KUKA KRL program: CIRCULO10X10_00.src

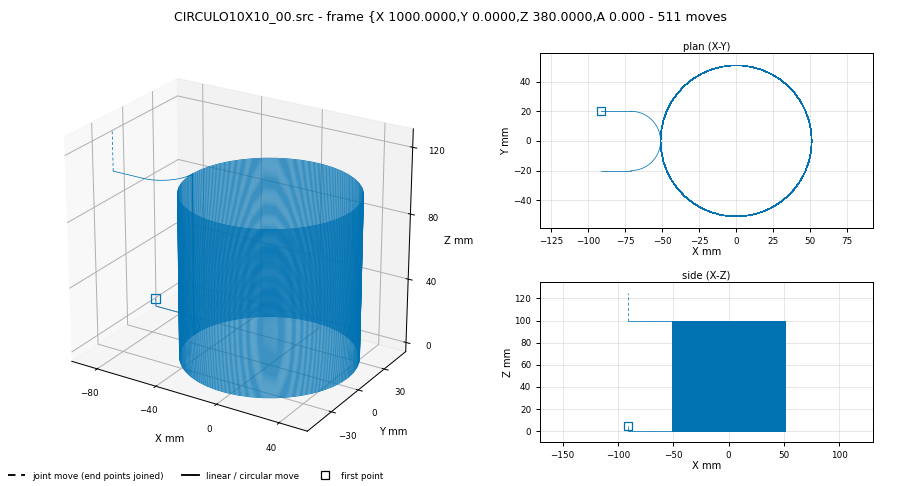
[picture p0: tool path of CIRCULO10X10_00.src in frame {X 1000.0000,Y 0.0000,Z 380.0000,A 0.000, 511 of 513 moves have a stored position in this frame; points joined in program order, loops and branches not executed]
&ACCESS RVP
&REL 1
&COMMENT GENERATED BY ROBOTMASTER
&PARAM TEMPLATE = C:\KRC\Roboter\Template\vorgabe
&PARAM EDITMASK = *
DEF CIRCULO10X2_00()

EXT BAS (BAS_COMMAND :IN,REAL :IN )

INT I

BAS (#INITMOV,0 )

;******SETTINGS FOR PTP MOTION***********************
;FOLD
;SET PTP $VEL_AXIS AND $ACC_AXIS
FOR I=1 TO 6
   $VEL_AXIS[I]=50
   $ACC_AXIS[I]=100
ENDFOR
;ENDFOLD (SET PTP $VEL_AXIS AND $ACC_AXIS)

;******SETTINGS FOR LIN AND ARC MOTION***************
;FOLD
;SET LIN AND ARC MOTION VARIABLES
$VEL.CP=0.262059
$VEL.ORI1=200
$VEL.ORI2=200
$ACC.ORI1=100
$ACC.ORI2=100
;ENDFOLD (SET LIN AND ARC MOTION VARIABLES)

;******SETTINGS FOR POSITIONING CRITERIA*************
;FOLD
;SET POSITIONING CRITERIA
  $APO.CDIS = 0.5000
  $ORI_TYPE = #VAR
;ENDFOLD (SET POSITIONING CRITERIA)

$BASE={X 1000.0000,Y 0.0000,Z 380.0000,A 0.0000,B 0.0000,C 0.0000}
$TOOL={X 63.3526,Y -0.0008,Z 236.7470,A 0.0000,B 30.5004,C 0.0000}

$ADVANCE = 5
PTP  {A1 20.0000,A2 -90.0000,A3 90.0000,A4 0.0000,A5 45.0000,A6 0.0000}
PTP  {X -91.0000,Y 20.0000,Z 5.0000,A 180.0000,B 0.0000,C 180.0000,S 2,T 35}
PTP  {X -91.0000,Y 20.0000,Z 2.0000,A 180.0000,B 0.0000,C 180.0000,S 2,T 35}
$VEL.CP=0.1  ;100mm/s
LIN  {X -91.0000,Y 20.0000,Z 0.0000,A 180.0000,B 0.0000,C 180.0000} C_DIS
LIN  {X -71.0000,Y 20.0000,Z 0.0000,A 180.0000,B 0.0000,C 180.0000} C_DIS
CIRC {X -56.8579,Y 14.1421,Z 0.0000,A 180.0000,B 0.0000,C 180.0000},{X -51.0000,Y 0.0000,Z 0.0000,A 180.0000,B 0.0000,C 180.0000} C_DIS
CIRC {X 0.0000,Y -51.0000,Z 0.0000,A 180.0000,B 0.0000,C 180.0000},{X 51.0000,Y 0.0000,Z 0.0000,A 180.0000,B 0.0000,C 180.0000} C_DIS
CIRC {X 0.0000,Y 51.0000,Z 0.0000,A 180.0000,B 0.0000,C 180.0000},{X -51.0000,Y 0.0000,Z 0.0000,A 180.0000,B 0.0000,C 180.0000} C_DIS
LIN  {X -51.0000,Y 0.0000,Z 0.5970,A 180.0000,B 0.0000,C 180.0000} C_DIS
CIRC {X 0.0000,Y -51.0000,Z 0.5970,A 180.0000,B 0.0000,C 180.0000},{X 51.0000,Y 0.0000,Z 0.5970,A 180.0000,B 0.0000,C 180.0000} C_DIS
CIRC {X 0.0000,Y 51.0000,Z 0.5970,A 180.0000,B 0.0000,C 180.0000},{X -51.0000,Y 0.0000,Z 0.5970,A 180.0000,B 0.0000,C 180.0000} C_DIS
LIN  {X -51.0000,Y 0.0000,Z 1.1976,A 180.0000,B 0.0000,C 180.0000} C_DIS
CIRC {X 0.0000,Y -51.0000,Z 1.1976,A 180.0000,B 0.0000,C 180.0000},{X 51.0000,Y 0.0000,Z 1.1976,A 180.0000,B 0.0000,C 180.0000} C_DIS
CIRC {X 0.0000,Y 51.0000,Z 1.1976,A 180.0000,B 0.0000,C 180.0000},{X -51.0000,Y 0.0000,Z 1.1976,A 180.0000,B 0.0000,C 180.0000} C_DIS
LIN  {X -51.0000,Y 0.0000,Z 1.7964,A 180.0000,B 0.0000,C 180.0000} C_DIS
CIRC {X 0.0000,Y -51.0000,Z 1.7964,A 180.0000,B 0.0000,C 180.0000},{X 51.0000,Y 0.0000,Z 1.7964,A 180.0000,B 0.0000,C 180.0000} C_DIS
CIRC {X 0.0000,Y 51.0000,Z 1.7964,A 180.0000,B 0.0000,C 180.0000},{X -51.0000,Y 0.0000,Z 1.7964,A 180.0000,B 0.0000,C 180.0000} C_DIS
LIN  {X -51.0000,Y 0.0000,Z 2.3952,A 180.0000,B 0.0000,C 180.0000} C_DIS
CIRC {X 0.0000,Y -51.0000,Z 2.3952,A 180.0000,B 0.0000,C 180.0000},{X 51.0000,Y 0.0000,Z 2.3952,A 180.0000,B 0.0000,C 180.0000} C_DIS
CIRC {X 0.0000,Y 51.0000,Z 2.3952,A 180.0000,B 0.0000,C 180.0000},{X -51.0000,Y 0.0000,Z 2.3952,A 180.0000,B 0.0000,C 180.0000} C_DIS
LIN  {X -51.0000,Y 0.0000,Z 2.9940,A 180.0000,B 0.0000,C 180.0000} C_DIS
CIRC {X 0.0000,Y -51.0000,Z 2.9940,A 180.0000,B 0.0000,C 180.0000},{X 51.0000,Y 0.0000,Z 2.9940,A 180.0000,B 0.0000,C 180.0000} C_DIS
CIRC {X 0.0000,Y 51.0000,Z 2.9940,A 180.0000,B 0.0000,C 180.0000},{X -51.0000,Y 0.0000,Z 2.9940,A 180.0000,B 0.0000,C 180.0000} C_DIS
LIN  {X -51.0000,Y 0.0000,Z 3.5928,A 180.0000,B 0.0000,C 180.0000} C_DIS
CIRC {X 0.0000,Y -51.0000,Z 3.5928,A 180.0000,B 0.0000,C 180.0000},{X 51.0000,Y 0.0000,Z 3.5928,A 180.0000,B 0.0000,C 180.0000} C_DIS
CIRC {X 0.0000,Y 51.0000,Z 3.5928,A 180.0000,B 0.0000,C 180.0000},{X -51.0000,Y 0.0000,Z 3.5928,A 180.0000,B 0.0000,C 180.0000} C_DIS
LIN  {X -51.0000,Y 0.0000,Z 4.1916,A 180.0000,B 0.0000,C 180.0000} C_DIS
CIRC {X 0.0000,Y -51.0000,Z 4.1916,A 180.0000,B 0.0000,C 180.0000},{X 51.0000,Y 0.0000,Z 4.1916,A 180.0000,B 0.0000,C 180.0000} C_DIS
CIRC {X 0.0000,Y 51.0000,Z 4.1916,A 180.0000,B 0.0000,C 180.0000},{X -51.0000,Y 0.0000,Z 4.1916,A 180.0000,B 0.0000,C 180.0000} C_DIS
LIN  {X -51.0000,Y 0.0000,Z 4.7904,A 180.0000,B 0.0000,C 180.0000} C_DIS
CIRC {X 0.0000,Y -51.0000,Z 4.7904,A 180.0000,B 0.0000,C 180.0000},{X 51.0000,Y 0.0000,Z 4.7904,A 180.0000,B 0.0000,C 180.0000} C_DIS
CIRC {X 0.0000,Y 51.0000,Z 4.7904,A 180.0000,B 0.0000,C 180.0000},{X -51.0000,Y 0.0000,Z 4.7904,A 180.0000,B 0.0000,C 180.0000} C_DIS
LIN  {X -51.0000,Y 0.0000,Z 5.3892,A 180.0000,B 0.0000,C 180.0000} C_DIS
CIRC {X 0.0000,Y -51.0000,Z 5.3892,A 180.0000,B 0.0000,C 180.0000},{X 51.0000,Y 0.0000,Z 5.3892,A 180.0000,B 0.0000,C 180.0000} C_DIS
CIRC {X 0.0000,Y 51.0000,Z 5.3892,A 180.0000,B 0.0000,C 180.0000},{X -51.0000,Y 0.0000,Z 5.3892,A 180.0000,B 0.0000,C 180.0000} C_DIS
LIN  {X -51.0000,Y 0.0000,Z 5.9880,A 180.0000,B 0.0000,C 180.0000} C_DIS
CIRC {X 0.0000,Y -51.0000,Z 5.9880,A 180.0000,B 0.0000,C 180.0000},{X 51.0000,Y 0.0000,Z 5.9880,A 180.0000,B 0.0000,C 180.0000} C_DIS
CIRC {X 0.0000,Y 51.0000,Z 5.9880,A 180.0000,B 0.0000,C 180.0000},{X -51.0000,Y 0.0000,Z 5.9880,A 180.0000,B 0.0000,C 180.0000} C_DIS
LIN  {X -51.0000,Y 0.0000,Z 6.5868,A 180.0000,B 0.0000,C 180.0000} C_DIS
CIRC {X 0.0000,Y -51.0000,Z 6.5868,A 180.0000,B 0.0000,C 180.0000},{X 51.0000,Y 0.0000,Z 6.5868,A 180.0000,B 0.0000,C 180.0000} C_DIS
CIRC {X 0.0000,Y 51.0000,Z 6.5868,A 180.0000,B 0.0000,C 180.0000},{X -51.0000,Y 0.0000,Z 6.5868,A 180.0000,B 0.0000,C 180.0000} C_DIS
LIN  {X -51.0000,Y 0.0000,Z 7.1856,A 180.0000,B 0.0000,C 180.0000} C_DIS
CIRC {X 0.0000,Y -51.0000,Z 7.1856,A 180.0000,B 0.0000,C 180.0000},{X 51.0000,Y 0.0000,Z 7.1856,A 180.0000,B 0.0000,C 180.0000} C_DIS
CIRC {X 0.0000,Y 51.0000,Z 7.1856,A 180.0000,B 0.0000,C 180.0000},{X -51.0000,Y 0.0000,Z 7.1856,A 180.0000,B 0.0000,C 180.0000} C_DIS
LIN  {X -51.0000,Y 0.0000,Z 7.7844,A 180.0000,B 0.0000,C 180.0000} C_DIS
CIRC {X 0.0000,Y -51.0000,Z 7.7844,A 180.0000,B 0.0000,C 180.0000},{X 51.0000,Y 0.0000,Z 7.7844,A 180.0000,B 0.0000,C 180.0000} C_DIS
CIRC {X 0.0000,Y 51.0000,Z 7.7844,A 180.0000,B 0.0000,C 180.0000},{X -51.0000,Y 0.0000,Z 7.7844,A 180.0000,B 0.0000,C 180.0000} C_DIS
LIN  {X -51.0000,Y 0.0000,Z 8.3832,A 180.0000,B 0.0000,C 180.0000} C_DIS
CIRC {X 0.0000,Y -51.0000,Z 8.3832,A 180.0000,B 0.0000,C 180.0000},{X 51.0000,Y 0.0000,Z 8.3832,A 180.0000,B 0.0000,C 180.0000} C_DIS
CIRC {X 0.0000,Y 51.0000,Z 8.3832,A 180.0000,B 0.0000,C 180.0000},{X -51.0000,Y 0.0000,Z 8.3832,A 180.0000,B 0.0000,C 180.0000} C_DIS
LIN  {X -51.0000,Y 0.0000,Z 8.9820,A 180.0000,B 0.0000,C 180.0000} C_DIS
CIRC {X 0.0000,Y -51.0000,Z 8.9820,A 180.0000,B 0.0000,C 180.0000},{X 51.0000,Y 0.0000,Z 8.9820,A 180.0000,B 0.0000,C 180.0000} C_DIS
CIRC {X 0.0000,Y 51.0000,Z 8.9820,A 180.0000,B 0.0000,C 180.0000},{X -51.0000,Y 0.0000,Z 8.9820,A 180.0000,B 0.0000,C 180.0000} C_DIS
LIN  {X -51.0000,Y 0.0000,Z 9.5808,A 180.0000,B 0.0000,C 180.0000} C_DIS
CIRC {X 0.0000,Y -51.0000,Z 9.5808,A 180.0000,B 0.0000,C 180.0000},{X 51.0000,Y 0.0000,Z 9.5808,A 180.0000,B 0.0000,C 180.0000} C_DIS
CIRC {X 0.0000,Y 51.0000,Z 9.5808,A 180.0000,B 0.0000,C 180.0000},{X -51.0000,Y 0.0000,Z 9.5808,A 180.0000,B 0.0000,C 180.0000} C_DIS
LIN  {X -51.0000,Y 0.0000,Z 10.1796,A 180.0000,B 0.0000,C 180.0000} C_DIS
CIRC {X 0.0000,Y -51.0000,Z 10.1796,A 180.0000,B 0.0000,C 180.0000},{X 51.0000,Y 0.0000,Z 10.1796,A 180.0000,B 0.0000,C 180.0000} C_DIS
CIRC {X 0.0000,Y 51.0000,Z 10.1796,A 180.0000,B 0.0000,C 180.0000},{X -51.0000,Y 0.0000,Z 10.1796,A 180.0000,B 0.0000,C 180.0000} C_DIS
LIN  {X -51.0000,Y 0.0000,Z 10.7784,A 180.0000,B 0.0000,C 180.0000} C_DIS
CIRC {X 0.0000,Y -51.0000,Z 10.7784,A 180.0000,B 0.0000,C 180.0000},{X 51.0000,Y 0.0000,Z 10.7784,A 180.0000,B 0.0000,C 180.0000} C_DIS
CIRC {X 0.0000,Y 51.0000,Z 10.7784,A 180.0000,B 0.0000,C 180.0000},{X -51.0000,Y 0.0000,Z 10.7784,A 180.0000,B 0.0000,C 180.0000} C_DIS
LIN  {X -51.0000,Y 0.0000,Z 11.3772,A 180.0000,B 0.0000,C 180.0000} C_DIS
CIRC {X 0.0000,Y -51.0000,Z 11.3772,A 180.0000,B 0.0000,C 180.0000},{X 51.0000,Y 0.0000,Z 11.3772,A 180.0000,B 0.0000,C 180.0000} C_DIS
CIRC {X 0.0000,Y 51.0000,Z 11.3772,A 180.0000,B 0.0000,C 180.0000},{X -51.0000,Y 0.0000,Z 11.3772,A 180.0000,B 0.0000,C 180.0000} C_DIS
LIN  {X -51.0000,Y 0.0000,Z 11.9760,A 180.0000,B 0.0000,C 180.0000} C_DIS
CIRC {X 0.0000,Y -51.0000,Z 11.9760,A 180.0000,B 0.0000,C 180.0000},{X 51.0000,Y 0.0000,Z 11.9760,A 180.0000,B 0.0000,C 180.0000} C_DIS
CIRC {X 0.0000,Y 51.0000,Z 11.9760,A 180.0000,B 0.0000,C 180.0000},{X -51.0000,Y 0.0000,Z 11.9760,A 180.0000,B 0.0000,C 180.0000} C_DIS
LIN  {X -51.0000,Y 0.0000,Z 12.5748,A 180.0000,B 0.0000,C 180.0000} C_DIS
CIRC {X 0.0000,Y -51.0000,Z 12.5748,A 180.0000,B 0.0000,C 180.0000},{X 51.0000,Y 0.0000,Z 12.5748,A 180.0000,B 0.0000,C 180.0000} C_DIS
CIRC {X 0.0000,Y 51.0000,Z 12.5748,A 180.0000,B 0.0000,C 180.0000},{X -51.0000,Y 0.0000,Z 12.5748,A 180.0000,B 0.0000,C 180.0000} C_DIS
LIN  {X -51.0000,Y 0.0000,Z 13.1737,A 180.0000,B 0.0000,C 180.0000} C_DIS
CIRC {X 0.0000,Y -51.0000,Z 13.1737,A 180.0000,B 0.0000,C 180.0000},{X 51.0000,Y 0.0000,Z 13.1737,A 180.0000,B 0.0000,C 180.0000} C_DIS
CIRC {X 0.0000,Y 51.0000,Z 13.1737,A 180.0000,B 0.0000,C 180.0000},{X -51.0000,Y 0.0000,Z 13.1737,A 180.0000,B 0.0000,C 180.0000} C_DIS
LIN  {X -51.0000,Y 0.0000,Z 13.7725,A 180.0000,B 0.0000,C 180.0000} C_DIS
CIRC {X 0.0000,Y -51.0000,Z 13.7725,A 180.0000,B 0.0000,C 180.0000},{X 51.0000,Y 0.0000,Z 13.7725,A 180.0000,B 0.0000,C 180.0000} C_DIS
CIRC {X 0.0000,Y 51.0000,Z 13.7725,A 180.0000,B 0.0000,C 180.0000},{X -51.0000,Y 0.0000,Z 13.7725,A 180.0000,B 0.0000,C 180.0000} C_DIS
LIN  {X -51.0000,Y 0.0000,Z 14.3713,A 180.0000,B 0.0000,C 180.0000} C_DIS
CIRC {X 0.0000,Y -51.0000,Z 14.3713,A 180.0000,B 0.0000,C 180.0000},{X 51.0000,Y 0.0000,Z 14.3713,A 180.0000,B 0.0000,C 180.0000} C_DIS
CIRC {X 0.0000,Y 51.0000,Z 14.3713,A 180.0000,B 0.0000,C 180.0000},{X -51.0000,Y 0.0000,Z 14.3713,A 180.0000,B 0.0000,C 180.0000} C_DIS
LIN  {X -51.0000,Y 0.0000,Z 14.9701,A 180.0000,B 0.0000,C 180.0000} C_DIS
CIRC {X 0.0000,Y -51.0000,Z 14.9701,A 180.0000,B 0.0000,C 180.0000},{X 51.0000,Y 0.0000,Z 14.9701,A 180.0000,B 0.0000,C 180.0000} C_DIS
CIRC {X 0.0000,Y 51.0000,Z 14.9701,A 180.0000,B 0.0000,C 180.0000},{X -51.0000,Y 0.0000,Z 14.9701,A 180.0000,B 0.0000,C 180.0000} C_DIS
LIN  {X -51.0000,Y 0.0000,Z 15.5689,A 180.0000,B 0.0000,C 180.0000} C_DIS
CIRC {X 0.0000,Y -51.0000,Z 15.5689,A 180.0000,B 0.0000,C 180.0000},{X 51.0000,Y 0.0000,Z 15.5689,A 180.0000,B 0.0000,C 180.0000} C_DIS
CIRC {X 0.0000,Y 51.0000,Z 15.5689,A 180.0000,B 0.0000,C 180.0000},{X -51.0000,Y 0.0000,Z 15.5689,A 180.0000,B 0.0000,C 180.0000} C_DIS
LIN  {X -51.0000,Y 0.0000,Z 16.1677,A 180.0000,B 0.0000,C 180.0000} C_DIS
CIRC {X 0.0000,Y -51.0000,Z 16.1677,A 180.0000,B 0.0000,C 180.0000},{X 51.0000,Y 0.0000,Z 16.1677,A 180.0000,B 0.0000,C 180.0000} C_DIS
CIRC {X 0.0000,Y 51.0000,Z 16.1677,A 180.0000,B 0.0000,C 180.0000},{X -51.0000,Y 0.0000,Z 16.1677,A 180.0000,B 0.0000,C 180.0000} C_DIS
LIN  {X -51.0000,Y 0.0000,Z 16.7665,A 180.0000,B 0.0000,C 180.0000} C_DIS
CIRC {X 0.0000,Y -51.0000,Z 16.7665,A 180.0000,B 0.0000,C 180.0000},{X 51.0000,Y 0.0000,Z 16.7665,A 180.0000,B 0.0000,C 180.0000} C_DIS
CIRC {X 0.0000,Y 51.0000,Z 16.7665,A 180.0000,B 0.0000,C 180.0000},{X -51.0000,Y 0.0000,Z 16.7665,A 180.0000,B 0.0000,C 180.0000} C_DIS
LIN  {X -51.0000,Y 0.0000,Z 17.3653,A 180.0000,B 0.0000,C 180.0000} C_DIS
CIRC {X 0.0000,Y -51.0000,Z 17.3653,A 180.0000,B 0.0000,C 180.0000},{X 51.0000,Y 0.0000,Z 17.3653,A 180.0000,B 0.0000,C 180.0000} C_DIS
CIRC {X 0.0000,Y 51.0000,Z 17.3653,A 180.0000,B 0.0000,C 180.0000},{X -51.0000,Y 0.0000,Z 17.3653,A 180.0000,B 0.0000,C 180.0000} C_DIS
LIN  {X -51.0000,Y 0.0000,Z 17.9641,A 180.0000,B 0.0000,C 180.0000} C_DIS
CIRC {X 0.0000,Y -51.0000,Z 17.9641,A 180.0000,B 0.0000,C 180.0000},{X 51.0000,Y 0.0000,Z 17.9641,A 180.0000,B 0.0000,C 180.0000} C_DIS
CIRC {X 0.0000,Y 51.0000,Z 17.9641,A 180.0000,B 0.0000,C 180.0000},{X -51.0000,Y 0.0000,Z 17.9641,A 180.0000,B 0.0000,C 180.0000} C_DIS
LIN  {X -51.0000,Y 0.0000,Z 18.5629,A 180.0000,B 0.0000,C 180.0000} C_DIS
CIRC {X 0.0000,Y -51.0000,Z 18.5629,A 180.0000,B 0.0000,C 180.0000},{X 51.0000,Y 0.0000,Z 18.5629,A 180.0000,B 0.0000,C 180.0000} C_DIS
CIRC {X 0.0000,Y 51.0000,Z 18.5629,A 180.0000,B 0.0000,C 180.0000},{X -51.0000,Y 0.0000,Z 18.5629,A 180.0000,B 0.0000,C 180.0000} C_DIS
LIN  {X -51.0000,Y 0.0000,Z 19.1617,A 180.0000,B 0.0000,C 180.0000} C_DIS
CIRC {X 0.0000,Y -51.0000,Z 19.1617,A 180.0000,B 0.0000,C 180.0000},{X 51.0000,Y 0.0000,Z 19.1617,A 180.0000,B 0.0000,C 180.0000} C_DIS
CIRC {X 0.0000,Y 51.0000,Z 19.1617,A 180.0000,B 0.0000,C 180.0000},{X -51.0000,Y 0.0000,Z 19.1617,A 180.0000,B 0.0000,C 180.0000} C_DIS
LIN  {X -51.0000,Y 0.0000,Z 19.7605,A 180.0000,B 0.0000,C 180.0000} C_DIS
CIRC {X 0.0000,Y -51.0000,Z 19.7605,A 180.0000,B 0.0000,C 180.0000},{X 51.0000,Y 0.0000,Z 19.7605,A 180.0000,B 0.0000,C 180.0000} C_DIS
CIRC {X 0.0000,Y 51.0000,Z 19.7605,A 180.0000,B 0.0000,C 180.0000},{X -51.0000,Y 0.0000,Z 19.7605,A 180.0000,B 0.0000,C 180.0000} C_DIS
LIN  {X -51.0000,Y 0.0000,Z 20.3593,A 180.0000,B 0.0000,C 180.0000} C_DIS
CIRC {X 0.0000,Y -51.0000,Z 20.3593,A 180.0000,B 0.0000,C 180.0000},{X 51.0000,Y 0.0000,Z 20.3593,A 180.0000,B 0.0000,C 180.0000} C_DIS
CIRC {X 0.0000,Y 51.0000,Z 20.3593,A 180.0000,B 0.0000,C 180.0000},{X -51.0000,Y 0.0000,Z 20.3593,A 180.0000,B 0.0000,C 180.0000} C_DIS
LIN  {X -51.0000,Y 0.0000,Z 20.9581,A 180.0000,B 0.0000,C 180.0000} C_DIS
CIRC {X 0.0000,Y -51.0000,Z 20.9581,A 180.0000,B 0.0000,C 180.0000},{X 51.0000,Y 0.0000,Z 20.9581,A 180.0000,B 0.0000,C 180.0000} C_DIS
CIRC {X 0.0000,Y 51.0000,Z 20.9581,A 180.0000,B 0.0000,C 180.0000},{X -51.0000,Y 0.0000,Z 20.9581,A 180.0000,B 0.0000,C 180.0000} C_DIS
LIN  {X -51.0000,Y 0.0000,Z 21.5569,A 180.0000,B 0.0000,C 180.0000} C_DIS
CIRC {X 0.0000,Y -51.0000,Z 21.5569,A 180.0000,B 0.0000,C 180.0000},{X 51.0000,Y 0.0000,Z 21.5569,A 180.0000,B 0.0000,C 180.0000} C_DIS
CIRC {X 0.0000,Y 51.0000,Z 21.5569,A 180.0000,B 0.0000,C 180.0000},{X -51.0000,Y 0.0000,Z 21.5569,A 180.0000,B 0.0000,C 180.0000} C_DIS
LIN  {X -51.0000,Y 0.0000,Z 22.1557,A 180.0000,B 0.0000,C 180.0000} C_DIS
CIRC {X 0.0000,Y -51.0000,Z 22.1557,A 180.0000,B 0.0000,C 180.0000},{X 51.0000,Y 0.0000,Z 22.1557,A 180.0000,B 0.0000,C 180.0000} C_DIS
CIRC {X 0.0000,Y 51.0000,Z 22.1557,A 180.0000,B 0.0000,C 180.0000},{X -51.0000,Y 0.0000,Z 22.1557,A 180.0000,B 0.0000,C 180.0000} C_DIS
LIN  {X -51.0000,Y 0.0000,Z 22.7545,A 180.0000,B 0.0000,C 180.0000} C_DIS
CIRC {X 0.0000,Y -51.0000,Z 22.7545,A 180.0000,B 0.0000,C 180.0000},{X 51.0000,Y 0.0000,Z 22.7545,A 180.0000,B 0.0000,C 180.0000} C_DIS
CIRC {X 0.0000,Y 51.0000,Z 22.7545,A 180.0000,B 0.0000,C 180.0000},{X -51.0000,Y 0.0000,Z 22.7545,A 180.0000,B 0.0000,C 180.0000} C_DIS
LIN  {X -51.0000,Y 0.0000,Z 23.3533,A 180.0000,B 0.0000,C 180.0000} C_DIS
CIRC {X 0.0000,Y -51.0000,Z 23.3533,A 180.0000,B 0.0000,C 180.0000},{X 51.0000,Y 0.0000,Z 23.3533,A 180.0000,B 0.0000,C 180.0000} C_DIS
CIRC {X 0.0000,Y 51.0000,Z 23.3533,A 180.0000,B 0.0000,C 180.0000},{X -51.0000,Y 0.0000,Z 23.3533,A 180.0000,B 0.0000,C 180.0000} C_DIS
LIN  {X -51.0000,Y 0.0000,Z 23.9521,A 180.0000,B 0.0000,C 180.0000} C_DIS
CIRC {X 0.0000,Y -51.0000,Z 23.9521,A 180.0000,B 0.0000,C 180.0000},{X 51.0000,Y 0.0000,Z 23.9521,A 180.0000,B 0.0000,C 180.0000} C_DIS
CIRC {X 0.0000,Y 51.0000,Z 23.9521,A 180.0000,B 0.0000,C 180.0000},{X -51.0000,Y 0.0000,Z 23.9521,A 180.0000,B 0.0000,C 180.0000} C_DIS
LIN  {X -51.0000,Y 0.0000,Z 24.5509,A 180.0000,B 0.0000,C 180.0000} C_DIS
CIRC {X 0.0000,Y -51.0000,Z 24.5509,A 180.0000,B 0.0000,C 180.0000},{X 51.0000,Y 0.0000,Z 24.5509,A 180.0000,B 0.0000,C 180.0000} C_DIS
CIRC {X 0.0000,Y 51.0000,Z 24.5509,A 180.0000,B 0.0000,C 180.0000},{X -51.0000,Y 0.0000,Z 24.5509,A 180.0000,B 0.0000,C 180.0000} C_DIS
LIN  {X -51.0000,Y 0.0000,Z 25.1497,A 180.0000,B 0.0000,C 180.0000} C_DIS
CIRC {X 0.0000,Y -51.0000,Z 25.1497,A 180.0000,B 0.0000,C 180.0000},{X 51.0000,Y 0.0000,Z 25.1497,A 180.0000,B 0.0000,C 180.0000} C_DIS
CIRC {X 0.0000,Y 51.0000,Z 25.1497,A 180.0000,B 0.0000,C 180.0000},{X -51.0000,Y 0.0000,Z 25.1497,A 180.0000,B 0.0000,C 180.0000} C_DIS
LIN  {X -51.0000,Y 0.0000,Z 25.7485,A 180.0000,B 0.0000,C 180.0000} C_DIS
CIRC {X 0.0000,Y -51.0000,Z 25.7485,A 180.0000,B 0.0000,C 180.0000},{X 51.0000,Y 0.0000,Z 25.7485,A 180.0000,B 0.0000,C 180.0000} C_DIS
CIRC {X 0.0000,Y 51.0000,Z 25.7485,A 180.0000,B 0.0000,C 180.0000},{X -51.0000,Y 0.0000,Z 25.7485,A 180.0000,B 0.0000,C 180.0000} C_DIS
LIN  {X -51.0000,Y 0.0000,Z 26.3473,A 180.0000,B 0.0000,C 180.0000} C_DIS
CIRC {X 0.0000,Y -51.0000,Z 26.3473,A 180.0000,B 0.0000,C 180.0000},{X 51.0000,Y 0.0000,Z 26.3473,A 180.0000,B 0.0000,C 180.0000} C_DIS
CIRC {X 0.0000,Y 51.0000,Z 26.3473,A 180.0000,B 0.0000,C 180.0000},{X -51.0000,Y 0.0000,Z 26.3473,A 180.0000,B 0.0000,C 180.0000} C_DIS
LIN  {X -51.0000,Y 0.0000,Z 26.9461,A 180.0000,B 0.0000,C 180.0000} C_DIS
CIRC {X 0.0000,Y -51.0000,Z 26.9461,A 180.0000,B 0.0000,C 180.0000},{X 51.0000,Y 0.0000,Z 26.9461,A 180.0000,B 0.0000,C 180.0000} C_DIS
CIRC {X 0.0000,Y 51.0000,Z 26.9461,A 180.0000,B 0.0000,C 180.0000},{X -51.0000,Y 0.0000,Z 26.9461,A 180.0000,B 0.0000,C 180.0000} C_DIS
LIN  {X -51.0000,Y 0.0000,Z 27.5449,A 180.0000,B 0.0000,C 180.0000} C_DIS
CIRC {X 0.0000,Y -51.0000,Z 27.5449,A 180.0000,B 0.0000,C 180.0000},{X 51.0000,Y 0.0000,Z 27.5449,A 180.0000,B 0.0000,C 180.0000} C_DIS
CIRC {X 0.0000,Y 51.0000,Z 27.5449,A 180.0000,B 0.0000,C 180.0000},{X -51.0000,Y 0.0000,Z 27.5449,A 180.0000,B 0.0000,C 180.0000} C_DIS
LIN  {X -51.0000,Y 0.0000,Z 28.1437,A 180.0000,B 0.0000,C 180.0000} C_DIS
CIRC {X 0.0000,Y -51.0000,Z 28.1437,A 180.0000,B 0.0000,C 180.0000},{X 51.0000,Y 0.0000,Z 28.1437,A 180.0000,B 0.0000,C 180.0000} C_DIS
CIRC {X 0.0000,Y 51.0000,Z 28.1437,A 180.0000,B 0.0000,C 180.0000},{X -51.0000,Y 0.0000,Z 28.1437,A 180.0000,B 0.0000,C 180.0000} C_DIS
LIN  {X -51.0000,Y 0.0000,Z 28.7425,A 180.0000,B 0.0000,C 180.0000} C_DIS
CIRC {X 0.0000,Y -51.0000,Z 28.7425,A 180.0000,B 0.0000,C 180.0000},{X 51.0000,Y 0.0000,Z 28.7425,A 180.0000,B 0.0000,C 180.0000} C_DIS
CIRC {X 0.0000,Y 51.0000,Z 28.7425,A 180.0000,B 0.0000,C 180.0000},{X -51.0000,Y 0.0000,Z 28.7425,A 180.0000,B 0.0000,C 180.0000} C_DIS
LIN  {X -51.0000,Y 0.0000,Z 29.3413,A 180.0000,B 0.0000,C 180.0000} C_DIS
CIRC {X 0.0000,Y -51.0000,Z 29.3413,A 180.0000,B 0.0000,C 180.0000},{X 51.0000,Y 0.0000,Z 29.3413,A 180.0000,B 0.0000,C 180.0000} C_DIS
CIRC {X 0.0000,Y 51.0000,Z 29.3413,A 180.0000,B 0.0000,C 180.0000},{X -51.0000,Y 0.0000,Z 29.3413,A 180.0000,B 0.0000,C 180.0000} C_DIS
LIN  {X -51.0000,Y 0.0000,Z 29.9401,A 180.0000,B 0.0000,C 180.0000} C_DIS
CIRC {X 0.0000,Y -51.0000,Z 29.9401,A 180.0000,B 0.0000,C 180.0000},{X 51.0000,Y 0.0000,Z 29.9401,A 180.0000,B 0.0000,C 180.0000} C_DIS
CIRC {X 0.0000,Y 51.0000,Z 29.9401,A 180.0000,B 0.0000,C 180.0000},{X -51.0000,Y 0.0000,Z 29.9401,A 180.0000,B 0.0000,C 180.0000} C_DIS
LIN  {X -51.0000,Y 0.0000,Z 30.5389,A 180.0000,B 0.0000,C 180.0000} C_DIS
CIRC {X 0.0000,Y -51.0000,Z 30.5389,A 180.0000,B 0.0000,C 180.0000},{X 51.0000,Y 0.0000,Z 30.5389,A 180.0000,B 0.0000,C 180.0000} C_DIS
CIRC {X 0.0000,Y 51.0000,Z 30.5389,A 180.0000,B 0.0000,C 180.0000},{X -51.0000,Y 0.0000,Z 30.5389,A 180.0000,B 0.0000,C 180.0000} C_DIS
LIN  {X -51.0000,Y 0.0000,Z 31.1377,A 180.0000,B 0.0000,C 180.0000} C_DIS
CIRC {X 0.0000,Y -51.0000,Z 31.1377,A 180.0000,B 0.0000,C 180.0000},{X 51.0000,Y 0.0000,Z 31.1377,A 180.0000,B 0.0000,C 180.0000} C_DIS
CIRC {X 0.0000,Y 51.0000,Z 31.1377,A 180.0000,B 0.0000,C 180.0000},{X -51.0000,Y 0.0000,Z 31.1377,A 180.0000,B 0.0000,C 180.0000} C_DIS
LIN  {X -51.0000,Y 0.0000,Z 31.7365,A 180.0000,B 0.0000,C 180.0000} C_DIS
CIRC {X 0.0000,Y -51.0000,Z 31.7365,A 180.0000,B 0.0000,C 180.0000},{X 51.0000,Y 0.0000,Z 31.7365,A 180.0000,B 0.0000,C 180.0000} C_DIS
CIRC {X 0.0000,Y 51.0000,Z 31.7365,A 180.0000,B 0.0000,C 180.0000},{X -51.0000,Y 0.0000,Z 31.7365,A 180.0000,B 0.0000,C 180.0000} C_DIS
LIN  {X -51.0000,Y 0.0000,Z 32.3353,A 180.0000,B 0.0000,C 180.0000} C_DIS
CIRC {X 0.0000,Y -51.0000,Z 32.3353,A 180.0000,B 0.0000,C 180.0000},{X 51.0000,Y 0.0000,Z 32.3353,A 180.0000,B 0.0000,C 180.0000} C_DIS
CIRC {X 0.0000,Y 51.0000,Z 32.3353,A 180.0000,B 0.0000,C 180.0000},{X -51.0000,Y 0.0000,Z 32.3353,A 180.0000,B 0.0000,C 180.0000} C_DIS
LIN  {X -51.0000,Y 0.0000,Z 32.9341,A 180.0000,B 0.0000,C 180.0000} C_DIS
CIRC {X 0.0000,Y -51.0000,Z 32.9341,A 180.0000,B 0.0000,C 180.0000},{X 51.0000,Y 0.0000,Z 32.9341,A 180.0000,B 0.0000,C 180.0000} C_DIS
CIRC {X 0.0000,Y 51.0000,Z 32.9341,A 180.0000,B 0.0000,C 180.0000},{X -51.0000,Y 0.0000,Z 32.9341,A 180.0000,B 0.0000,C 180.0000} C_DIS
LIN  {X -51.0000,Y 0.0000,Z 33.5329,A 180.0000,B 0.0000,C 180.0000} C_DIS
CIRC {X 0.0000,Y -51.0000,Z 33.5329,A 180.0000,B 0.0000,C 180.0000},{X 51.0000,Y 0.0000,Z 33.5329,A 180.0000,B 0.0000,C 180.0000} C_DIS
CIRC {X 0.0000,Y 51.0000,Z 33.5329,A 180.0000,B 0.0000,C 180.0000},{X -51.0000,Y 0.0000,Z 33.5329,A 180.0000,B 0.0000,C 180.0000} C_DIS
LIN  {X -51.0000,Y 0.0000,Z 34.1317,A 180.0000,B 0.0000,C 180.0000} C_DIS
CIRC {X 0.0000,Y -51.0000,Z 34.1317,A 180.0000,B 0.0000,C 180.0000},{X 51.0000,Y 0.0000,Z 34.1317,A 180.0000,B 0.0000,C 180.0000} C_DIS
CIRC {X 0.0000,Y 51.0000,Z 34.1317,A 180.0000,B 0.0000,C 180.0000},{X -51.0000,Y 0.0000,Z 34.1317,A 180.0000,B 0.0000,C 180.0000} C_DIS
LIN  {X -51.0000,Y 0.0000,Z 34.7305,A 180.0000,B 0.0000,C 180.0000} C_DIS
CIRC {X 0.0000,Y -51.0000,Z 34.7305,A 180.0000,B 0.0000,C 180.0000},{X 51.0000,Y 0.0000,Z 34.7305,A 180.0000,B 0.0000,C 180.0000} C_DIS
CIRC {X 0.0000,Y 51.0000,Z 34.7305,A 180.0000,B 0.0000,C 180.0000},{X -51.0000,Y 0.0000,Z 34.7305,A 180.0000,B 0.0000,C 180.0000} C_DIS
LIN  {X -51.0000,Y 0.0000,Z 35.3293,A 180.0000,B 0.0000,C 180.0000} C_DIS
CIRC {X 0.0000,Y -51.0000,Z 35.3293,A 180.0000,B 0.0000,C 180.0000},{X 51.0000,Y 0.0000,Z 35.3293,A 180.0000,B 0.0000,C 180.0000} C_DIS
CIRC {X 0.0000,Y 51.0000,Z 35.3293,A 180.0000,B 0.0000,C 180.0000},{X -51.0000,Y 0.0000,Z 35.3293,A 180.0000,B 0.0000,C 180.0000} C_DIS
LIN  {X -51.0000,Y 0.0000,Z 35.9281,A 180.0000,B 0.0000,C 180.0000} C_DIS
CIRC {X 0.0000,Y -51.0000,Z 35.9281,A 180.0000,B 0.0000,C 180.0000},{X 51.0000,Y 0.0000,Z 35.9281,A 180.0000,B 0.0000,C 180.0000} C_DIS
CIRC {X 0.0000,Y 51.0000,Z 35.9281,A 180.0000,B 0.0000,C 180.0000},{X -51.0000,Y 0.0000,Z 35.9281,A 180.0000,B 0.0000,C 180.0000} C_DIS
LIN  {X -51.0000,Y 0.0000,Z 36.5269,A 180.0000,B 0.0000,C 180.0000} C_DIS
CIRC {X 0.0000,Y -51.0000,Z 36.5269,A 180.0000,B 0.0000,C 180.0000},{X 51.0000,Y 0.0000,Z 36.5269,A 180.0000,B 0.0000,C 180.0000} C_DIS
CIRC {X 0.0000,Y 51.0000,Z 36.5269,A 180.0000,B 0.0000,C 180.0000},{X -51.0000,Y 0.0000,Z 36.5269,A 180.0000,B 0.0000,C 180.0000} C_DIS
LIN  {X -51.0000,Y 0.0000,Z 37.1257,A 180.0000,B 0.0000,C 180.0000} C_DIS
CIRC {X 0.0000,Y -51.0000,Z 37.1257,A 180.0000,B 0.0000,C 180.0000},{X 51.0000,Y 0.0000,Z 37.1257,A 180.0000,B 0.0000,C 180.0000} C_DIS
CIRC {X 0.0000,Y 51.0000,Z 37.1257,A 180.0000,B 0.0000,C 180.0000},{X -51.0000,Y 0.0000,Z 37.1257,A 180.0000,B 0.0000,C 180.0000} C_DIS
LIN  {X -51.0000,Y 0.0000,Z 37.7246,A 180.0000,B 0.0000,C 180.0000} C_DIS
CIRC {X 0.0000,Y -51.0000,Z 37.7246,A 180.0000,B 0.0000,C 180.0000},{X 51.0000,Y 0.0000,Z 37.7246,A 180.0000,B 0.0000,C 180.0000} C_DIS
CIRC {X 0.0000,Y 51.0000,Z 37.7246,A 180.0000,B 0.0000,C 180.0000},{X -51.0000,Y 0.0000,Z 37.7246,A 180.0000,B 0.0000,C 180.0000} C_DIS
LIN  {X -51.0000,Y 0.0000,Z 38.3234,A 180.0000,B 0.0000,C 180.0000} C_DIS
CIRC {X 0.0000,Y -51.0000,Z 38.3234,A 180.0000,B 0.0000,C 180.0000},{X 51.0000,Y 0.0000,Z 38.3234,A 180.0000,B 0.0000,C 180.0000} C_DIS
CIRC {X 0.0000,Y 51.0000,Z 38.3234,A 180.0000,B 0.0000,C 180.0000},{X -51.0000,Y 0.0000,Z 38.3234,A 180.0000,B 0.0000,C 180.0000} C_DIS
LIN  {X -51.0000,Y 0.0000,Z 38.9222,A 180.0000,B 0.0000,C 180.0000} C_DIS
CIRC {X 0.0000,Y -51.0000,Z 38.9222,A 180.0000,B 0.0000,C 180.0000},{X 51.0000,Y 0.0000,Z 38.9222,A 180.0000,B 0.0000,C 180.0000} C_DIS
CIRC {X 0.0000,Y 51.0000,Z 38.9222,A 180.0000,B 0.0000,C 180.0000},{X -51.0000,Y 0.0000,Z 38.9222,A 180.0000,B 0.0000,C 180.0000} C_DIS
LIN  {X -51.0000,Y 0.0000,Z 39.5210,A 180.0000,B 0.0000,C 180.0000} C_DIS
CIRC {X 0.0000,Y -51.0000,Z 39.5210,A 180.0000,B 0.0000,C 180.0000},{X 51.0000,Y 0.0000,Z 39.5210,A 180.0000,B 0.0000,C 180.0000} C_DIS
CIRC {X 0.0000,Y 51.0000,Z 39.5210,A 180.0000,B 0.0000,C 180.0000},{X -51.0000,Y 0.0000,Z 39.5210,A 180.0000,B 0.0000,C 180.0000} C_DIS
LIN  {X -51.0000,Y 0.0000,Z 40.1198,A 180.0000,B 0.0000,C 180.0000} C_DIS
CIRC {X 0.0000,Y -51.0000,Z 40.1198,A 180.0000,B 0.0000,C 180.0000},{X 51.0000,Y 0.0000,Z 40.1198,A 180.0000,B 0.0000,C 180.0000} C_DIS
CIRC {X 0.0000,Y 51.0000,Z 40.1198,A 180.0000,B 0.0000,C 180.0000},{X -51.0000,Y 0.0000,Z 40.1198,A 180.0000,B 0.0000,C 180.0000} C_DIS
LIN  {X -51.0000,Y 0.0000,Z 40.7186,A 180.0000,B 0.0000,C 180.0000} C_DIS
CIRC {X 0.0000,Y -51.0000,Z 40.7186,A 180.0000,B 0.0000,C 180.0000},{X 51.0000,Y 0.0000,Z 40.7186,A 180.0000,B 0.0000,C 180.0000} C_DIS
CIRC {X 0.0000,Y 51.0000,Z 40.7186,A 180.0000,B 0.0000,C 180.0000},{X -51.0000,Y 0.0000,Z 40.7186,A 180.0000,B 0.0000,C 180.0000} C_DIS
LIN  {X -51.0000,Y 0.0000,Z 41.3174,A 180.0000,B 0.0000,C 180.0000} C_DIS
CIRC {X 0.0000,Y -51.0000,Z 41.3174,A 180.0000,B 0.0000,C 180.0000},{X 51.0000,Y 0.0000,Z 41.3174,A 180.0000,B 0.0000,C 180.0000} C_DIS
CIRC {X 0.0000,Y 51.0000,Z 41.3174,A 180.0000,B 0.0000,C 180.0000},{X -51.0000,Y 0.0000,Z 41.3174,A 180.0000,B 0.0000,C 180.0000} C_DIS
LIN  {X -51.0000,Y 0.0000,Z 41.9162,A 180.0000,B 0.0000,C 180.0000} C_DIS
CIRC {X 0.0000,Y -51.0000,Z 41.9162,A 180.0000,B 0.0000,C 180.0000},{X 51.0000,Y 0.0000,Z 41.9162,A 180.0000,B 0.0000,C 180.0000} C_DIS
CIRC {X 0.0000,Y 51.0000,Z 41.9162,A 180.0000,B 0.0000,C 180.0000},{X -51.0000,Y 0.0000,Z 41.9162,A 180.0000,B 0.0000,C 180.0000} C_DIS
LIN  {X -51.0000,Y 0.0000,Z 42.5150,A 180.0000,B 0.0000,C 180.0000} C_DIS
CIRC {X 0.0000,Y -51.0000,Z 42.5150,A 180.0000,B 0.0000,C 180.0000},{X 51.0000,Y 0.0000,Z 42.5150,A 180.0000,B 0.0000,C 180.0000} C_DIS
CIRC {X 0.0000,Y 51.0000,Z 42.5150,A 180.0000,B 0.0000,C 180.0000},{X -51.0000,Y 0.0000,Z 42.5150,A 180.0000,B 0.0000,C 180.0000} C_DIS
LIN  {X -51.0000,Y 0.0000,Z 43.1138,A 180.0000,B 0.0000,C 180.0000} C_DIS
CIRC {X 0.0000,Y -51.0000,Z 43.1138,A 180.0000,B 0.0000,C 180.0000},{X 51.0000,Y 0.0000,Z 43.1138,A 180.0000,B 0.0000,C 180.0000} C_DIS
CIRC {X 0.0000,Y 51.0000,Z 43.1138,A 180.0000,B 0.0000,C 180.0000},{X -51.0000,Y 0.0000,Z 43.1138,A 180.0000,B 0.0000,C 180.0000} C_DIS
LIN  {X -51.0000,Y 0.0000,Z 43.7126,A 180.0000,B 0.0000,C 180.0000} C_DIS
CIRC {X 0.0000,Y -51.0000,Z 43.7126,A 180.0000,B 0.0000,C 180.0000},{X 51.0000,Y 0.0000,Z 43.7126,A 180.0000,B 0.0000,C 180.0000} C_DIS
CIRC {X 0.0000,Y 51.0000,Z 43.7126,A 180.0000,B 0.0000,C 180.0000},{X -51.0000,Y 0.0000,Z 43.7126,A 180.0000,B 0.0000,C 180.0000} C_DIS
LIN  {X -51.0000,Y 0.0000,Z 44.3114,A 180.0000,B 0.0000,C 180.0000} C_DIS
CIRC {X 0.0000,Y -51.0000,Z 44.3114,A 180.0000,B 0.0000,C 180.0000},{X 51.0000,Y 0.0000,Z 44.3114,A 180.0000,B 0.0000,C 180.0000} C_DIS
CIRC {X 0.0000,Y 51.0000,Z 44.3114,A 180.0000,B 0.0000,C 180.0000},{X -51.0000,Y 0.0000,Z 44.3114,A 180.0000,B 0.0000,C 180.0000} C_DIS
LIN  {X -51.0000,Y 0.0000,Z 44.9102,A 180.0000,B 0.0000,C 180.0000} C_DIS
CIRC {X 0.0000,Y -51.0000,Z 44.9102,A 180.0000,B 0.0000,C 180.0000},{X 51.0000,Y 0.0000,Z 44.9102,A 180.0000,B 0.0000,C 180.0000} C_DIS
CIRC {X 0.0000,Y 51.0000,Z 44.9102,A 180.0000,B 0.0000,C 180.0000},{X -51.0000,Y 0.0000,Z 44.9102,A 180.0000,B 0.0000,C 180.0000} C_DIS
LIN  {X -51.0000,Y 0.0000,Z 45.5090,A 180.0000,B 0.0000,C 180.0000} C_DIS
CIRC {X 0.0000,Y -51.0000,Z 45.5090,A 180.0000,B 0.0000,C 180.0000},{X 51.0000,Y 0.0000,Z 45.5090,A 180.0000,B 0.0000,C 180.0000} C_DIS
CIRC {X 0.0000,Y 51.0000,Z 45.5090,A 180.0000,B 0.0000,C 180.0000},{X -51.0000,Y 0.0000,Z 45.5090,A 180.0000,B 0.0000,C 180.0000} C_DIS
LIN  {X -51.0000,Y 0.0000,Z 46.1078,A 180.0000,B 0.0000,C 180.0000} C_DIS
CIRC {X 0.0000,Y -51.0000,Z 46.1078,A 180.0000,B 0.0000,C 180.0000},{X 51.0000,Y 0.0000,Z 46.1078,A 180.0000,B 0.0000,C 180.0000} C_DIS
CIRC {X 0.0000,Y 51.0000,Z 46.1078,A 180.0000,B 0.0000,C 180.0000},{X -51.0000,Y 0.0000,Z 46.1078,A 180.0000,B 0.0000,C 180.0000} C_DIS
LIN  {X -51.0000,Y 0.0000,Z 46.7066,A 180.0000,B 0.0000,C 180.0000} C_DIS
CIRC {X 0.0000,Y -51.0000,Z 46.7066,A 180.0000,B 0.0000,C 180.0000},{X 51.0000,Y 0.0000,Z 46.7066,A 180.0000,B 0.0000,C 180.0000} C_DIS
CIRC {X 0.0000,Y 51.0000,Z 46.7066,A 180.0000,B 0.0000,C 180.0000},{X -51.0000,Y 0.0000,Z 46.7066,A 180.0000,B 0.0000,C 180.0000} C_DIS
LIN  {X -51.0000,Y 0.0000,Z 47.3054,A 180.0000,B 0.0000,C 180.0000} C_DIS
CIRC {X 0.0000,Y -51.0000,Z 47.3054,A 180.0000,B 0.0000,C 180.0000},{X 51.0000,Y 0.0000,Z 47.3054,A 180.0000,B 0.0000,C 180.0000} C_DIS
CIRC {X 0.0000,Y 51.0000,Z 47.3054,A 180.0000,B 0.0000,C 180.0000},{X -51.0000,Y 0.0000,Z 47.3054,A 180.0000,B 0.0000,C 180.0000} C_DIS
LIN  {X -51.0000,Y 0.0000,Z 47.9042,A 180.0000,B 0.0000,C 180.0000} C_DIS
CIRC {X 0.0000,Y -51.0000,Z 47.9042,A 180.0000,B 0.0000,C 180.0000},{X 51.0000,Y 0.0000,Z 47.9042,A 180.0000,B 0.0000,C 180.0000} C_DIS
CIRC {X 0.0000,Y 51.0000,Z 47.9042,A 180.0000,B 0.0000,C 180.0000},{X -51.0000,Y 0.0000,Z 47.9042,A 180.0000,B 0.0000,C 180.0000} C_DIS
LIN  {X -51.0000,Y 0.0000,Z 48.5030,A 180.0000,B 0.0000,C 180.0000} C_DIS
CIRC {X 0.0000,Y -51.0000,Z 48.5030,A 180.0000,B 0.0000,C 180.0000},{X 51.0000,Y 0.0000,Z 48.5030,A 180.0000,B 0.0000,C 180.0000} C_DIS
CIRC {X 0.0000,Y 51.0000,Z 48.5030,A 180.0000,B 0.0000,C 180.0000},{X -51.0000,Y 0.0000,Z 48.5030,A 180.0000,B 0.0000,C 180.0000} C_DIS
LIN  {X -51.0000,Y 0.0000,Z 49.1018,A 180.0000,B 0.0000,C 180.0000} C_DIS
CIRC {X 0.0000,Y -51.0000,Z 49.1018,A 180.0000,B 0.0000,C 180.0000},{X 51.0000,Y 0.0000,Z 49.1018,A 180.0000,B 0.0000,C 180.0000} C_DIS
CIRC {X 0.0000,Y 51.0000,Z 49.1018,A 180.0000,B 0.0000,C 180.0000},{X -51.0000,Y 0.0000,Z 49.1018,A 180.0000,B 0.0000,C 180.0000} C_DIS
LIN  {X -51.0000,Y 0.0000,Z 49.7006,A 180.0000,B 0.0000,C 180.0000} C_DIS
CIRC {X 0.0000,Y -51.0000,Z 49.7006,A 180.0000,B 0.0000,C 180.0000},{X 51.0000,Y 0.0000,Z 49.7006,A 180.0000,B 0.0000,C 180.0000} C_DIS
CIRC {X 0.0000,Y 51.0000,Z 49.7006,A 180.0000,B 0.0000,C 180.0000},{X -51.0000,Y 0.0000,Z 49.7006,A 180.0000,B 0.0000,C 180.0000} C_DIS
LIN  {X -51.0000,Y 0.0000,Z 50.2994,A 180.0000,B 0.0000,C 180.0000} C_DIS
CIRC {X 0.0000,Y -51.0000,Z 50.2994,A 180.0000,B 0.0000,C 180.0000},{X 51.0000,Y 0.0000,Z 50.2994,A 180.0000,B 0.0000,C 180.0000} C_DIS
CIRC {X 0.0000,Y 51.0000,Z 50.2994,A 180.0000,B 0.0000,C 180.0000},{X -51.0000,Y 0.0000,Z 50.2994,A 180.0000,B 0.0000,C 180.0000} C_DIS
LIN  {X -51.0000,Y 0.0000,Z 50.8982,A 180.0000,B 0.0000,C 180.0000} C_DIS
CIRC {X 0.0000,Y -51.0000,Z 50.8982,A 180.0000,B 0.0000,C 180.0000},{X 51.0000,Y 0.0000,Z 50.8982,A 180.0000,B 0.0000,C 180.0000} C_DIS
CIRC {X 0.0000,Y 51.0000,Z 50.8982,A 180.0000,B 0.0000,C 180.0000},{X -51.0000,Y 0.0000,Z 50.8982,A 180.0000,B 0.0000,C 180.0000} C_DIS
LIN  {X -51.0000,Y 0.0000,Z 51.4970,A 180.0000,B 0.0000,C 180.0000} C_DIS
CIRC {X 0.0000,Y -51.0000,Z 51.4970,A 180.0000,B 0.0000,C 180.0000},{X 51.0000,Y 0.0000,Z 51.4970,A 180.0000,B 0.0000,C 180.0000} C_DIS
CIRC {X 0.0000,Y 51.0000,Z 51.4970,A 180.0000,B 0.0000,C 180.0000},{X -51.0000,Y 0.0000,Z 51.4970,A 180.0000,B 0.0000,C 180.0000} C_DIS
LIN  {X -51.0000,Y 0.0000,Z 52.0958,A 180.0000,B 0.0000,C 180.0000} C_DIS
CIRC {X 0.0000,Y -51.0000,Z 52.0958,A 180.0000,B 0.0000,C 180.0000},{X 51.0000,Y 0.0000,Z 52.0958,A 180.0000,B 0.0000,C 180.0000} C_DIS
CIRC {X 0.0000,Y 51.0000,Z 52.0958,A 180.0000,B 0.0000,C 180.0000},{X -51.0000,Y 0.0000,Z 52.0958,A 180.0000,B 0.0000,C 180.0000} C_DIS
LIN  {X -51.0000,Y 0.0000,Z 52.6946,A 180.0000,B 0.0000,C 180.0000} C_DIS
CIRC {X 0.0000,Y -51.0000,Z 52.6946,A 180.0000,B 0.0000,C 180.0000},{X 51.0000,Y 0.0000,Z 52.6946,A 180.0000,B 0.0000,C 180.0000} C_DIS
CIRC {X 0.0000,Y 51.0000,Z 52.6946,A 180.0000,B 0.0000,C 180.0000},{X -51.0000,Y 0.0000,Z 52.6946,A 180.0000,B 0.0000,C 180.0000} C_DIS
LIN  {X -51.0000,Y 0.0000,Z 53.2934,A 180.0000,B 0.0000,C 180.0000} C_DIS
CIRC {X 0.0000,Y -51.0000,Z 53.2934,A 180.0000,B 0.0000,C 180.0000},{X 51.0000,Y 0.0000,Z 53.2934,A 180.0000,B 0.0000,C 180.0000} C_DIS
CIRC {X 0.0000,Y 51.0000,Z 53.2934,A 180.0000,B 0.0000,C 180.0000},{X -51.0000,Y 0.0000,Z 53.2934,A 180.0000,B 0.0000,C 180.0000} C_DIS
LIN  {X -51.0000,Y 0.0000,Z 53.8922,A 180.0000,B 0.0000,C 180.0000} C_DIS
CIRC {X 0.0000,Y -51.0000,Z 53.8922,A 180.0000,B 0.0000,C 180.0000},{X 51.0000,Y 0.0000,Z 53.8922,A 180.0000,B 0.0000,C 180.0000} C_DIS
CIRC {X 0.0000,Y 51.0000,Z 53.8922,A 180.0000,B 0.0000,C 180.0000},{X -51.0000,Y 0.0000,Z 53.8922,A 180.0000,B 0.0000,C 180.0000} C_DIS
LIN  {X -51.0000,Y 0.0000,Z 54.4910,A 180.0000,B 0.0000,C 180.0000} C_DIS
CIRC {X 0.0000,Y -51.0000,Z 54.4910,A 180.0000,B 0.0000,C 180.0000},{X 51.0000,Y 0.0000,Z 54.4910,A 180.0000,B 0.0000,C 180.0000} C_DIS
CIRC {X 0.0000,Y 51.0000,Z 54.4910,A 180.0000,B 0.0000,C 180.0000},{X -51.0000,Y 0.0000,Z 54.4910,A 180.0000,B 0.0000,C 180.0000} C_DIS
LIN  {X -51.0000,Y 0.0000,Z 55.0898,A 180.0000,B 0.0000,C 180.0000} C_DIS
CIRC {X 0.0000,Y -51.0000,Z 55.0898,A 180.0000,B 0.0000,C 180.0000},{X 51.0000,Y 0.0000,Z 55.0898,A 180.0000,B 0.0000,C 180.0000} C_DIS
CIRC {X 0.0000,Y 51.0000,Z 55.0898,A 180.0000,B 0.0000,C 180.0000},{X -51.0000,Y 0.0000,Z 55.0898,A 180.0000,B 0.0000,C 180.0000} C_DIS
LIN  {X -51.0000,Y 0.0000,Z 55.6886,A 180.0000,B 0.0000,C 180.0000} C_DIS
CIRC {X 0.0000,Y -51.0000,Z 55.6886,A 180.0000,B 0.0000,C 180.0000},{X 51.0000,Y 0.0000,Z 55.6886,A 180.0000,B 0.0000,C 180.0000} C_DIS
CIRC {X 0.0000,Y 51.0000,Z 55.6886,A 180.0000,B 0.0000,C 180.0000},{X -51.0000,Y 0.0000,Z 55.6886,A 180.0000,B 0.0000,C 180.0000} C_DIS
LIN  {X -51.0000,Y 0.0000,Z 56.2874,A 180.0000,B 0.0000,C 180.0000} C_DIS
CIRC {X 0.0000,Y -51.0000,Z 56.2874,A 180.0000,B 0.0000,C 180.0000},{X 51.0000,Y 0.0000,Z 56.2874,A 180.0000,B 0.0000,C 180.0000} C_DIS
CIRC {X 0.0000,Y 51.0000,Z 56.2874,A 180.0000,B 0.0000,C 180.0000},{X -51.0000,Y 0.0000,Z 56.2874,A 180.0000,B 0.0000,C 180.0000} C_DIS
LIN  {X -51.0000,Y 0.0000,Z 56.8862,A 180.0000,B 0.0000,C 180.0000} C_DIS
CIRC {X 0.0000,Y -51.0000,Z 56.8862,A 180.0000,B 0.0000,C 180.0000},{X 51.0000,Y 0.0000,Z 56.8862,A 180.0000,B 0.0000,C 180.0000} C_DIS
CIRC {X 0.0000,Y 51.0000,Z 56.8862,A 180.0000,B 0.0000,C 180.0000},{X -51.0000,Y 0.0000,Z 56.8862,A 180.0000,B 0.0000,C 180.0000} C_DIS
LIN  {X -51.0000,Y 0.0000,Z 57.4850,A 180.0000,B 0.0000,C 180.0000} C_DIS
CIRC {X 0.0000,Y -51.0000,Z 57.4850,A 180.0000,B 0.0000,C 180.0000},{X 51.0000,Y 0.0000,Z 57.4850,A 180.0000,B 0.0000,C 180.0000} C_DIS
CIRC {X 0.0000,Y 51.0000,Z 57.4850,A 180.0000,B 0.0000,C 180.0000},{X -51.0000,Y 0.0000,Z 57.4850,A 180.0000,B 0.0000,C 180.0000} C_DIS
LIN  {X -51.0000,Y 0.0000,Z 58.0838,A 180.0000,B 0.0000,C 180.0000} C_DIS
CIRC {X 0.0000,Y -51.0000,Z 58.0838,A 180.0000,B 0.0000,C 180.0000},{X 51.0000,Y 0.0000,Z 58.0838,A 180.0000,B 0.0000,C 180.0000} C_DIS
CIRC {X 0.0000,Y 51.0000,Z 58.0838,A 180.0000,B 0.0000,C 180.0000},{X -51.0000,Y 0.0000,Z 58.0838,A 180.0000,B 0.0000,C 180.0000} C_DIS
LIN  {X -51.0000,Y 0.0000,Z 58.6826,A 180.0000,B 0.0000,C 180.0000} C_DIS
CIRC {X 0.0000,Y -51.0000,Z 58.6826,A 180.0000,B 0.0000,C 180.0000},{X 51.0000,Y 0.0000,Z 58.6826,A 180.0000,B 0.0000,C 180.0000} C_DIS
CIRC {X 0.0000,Y 51.0000,Z 58.6826,A 180.0000,B 0.0000,C 180.0000},{X -51.0000,Y 0.0000,Z 58.6826,A 180.0000,B 0.0000,C 180.0000} C_DIS
LIN  {X -51.0000,Y 0.0000,Z 59.2814,A 180.0000,B 0.0000,C 180.0000} C_DIS
CIRC {X 0.0000,Y -51.0000,Z 59.2814,A 180.0000,B 0.0000,C 180.0000},{X 51.0000,Y 0.0000,Z 59.2814,A 180.0000,B 0.0000,C 180.0000} C_DIS
CIRC {X 0.0000,Y 51.0000,Z 59.2814,A 180.0000,B 0.0000,C 180.0000},{X -51.0000,Y 0.0000,Z 59.2814,A 180.0000,B 0.0000,C 180.0000} C_DIS
LIN  {X -51.0000,Y 0.0000,Z 59.8802,A 180.0000,B 0.0000,C 180.0000} C_DIS
CIRC {X 0.0000,Y -51.0000,Z 59.8802,A 180.0000,B 0.0000,C 180.0000},{X 51.0000,Y 0.0000,Z 59.8802,A 180.0000,B 0.0000,C 180.0000} C_DIS
CIRC {X 0.0000,Y 51.0000,Z 59.8802,A 180.0000,B 0.0000,C 180.0000},{X -51.0000,Y 0.0000,Z 59.8802,A 180.0000,B 0.0000,C 180.0000} C_DIS
LIN  {X -51.0000,Y 0.0000,Z 60.4790,A 180.0000,B 0.0000,C 180.0000} C_DIS
CIRC {X 0.0000,Y -51.0000,Z 60.4790,A 180.0000,B 0.0000,C 180.0000},{X 51.0000,Y 0.0000,Z 60.4790,A 180.0000,B 0.0000,C 180.0000} C_DIS
CIRC {X 0.0000,Y 51.0000,Z 60.4790,A 180.0000,B 0.0000,C 180.0000},{X -51.0000,Y 0.0000,Z 60.4790,A 180.0000,B 0.0000,C 180.0000} C_DIS
LIN  {X -51.0000,Y 0.0000,Z 61.0778,A 180.0000,B 0.0000,C 180.0000} C_DIS
CIRC {X 0.0000,Y -51.0000,Z 61.0778,A 180.0000,B 0.0000,C 180.0000},{X 51.0000,Y 0.0000,Z 61.0778,A 180.0000,B 0.0000,C 180.0000} C_DIS
CIRC {X 0.0000,Y 51.0000,Z 61.0778,A 180.0000,B 0.0000,C 180.0000},{X -51.0000,Y 0.0000,Z 61.0778,A 180.0000,B 0.0000,C 180.0000} C_DIS
LIN  {X -51.0000,Y 0.0000,Z 61.6766,A 180.0000,B 0.0000,C 180.0000} C_DIS
CIRC {X 0.0000,Y -51.0000,Z 61.6766,A 180.0000,B 0.0000,C 180.0000},{X 51.0000,Y 0.0000,Z 61.6766,A 180.0000,B 0.0000,C 180.0000} C_DIS
CIRC {X 0.0000,Y 51.0000,Z 61.6766,A 180.0000,B 0.0000,C 180.0000},{X -51.0000,Y 0.0000,Z 61.6766,A 180.0000,B 0.0000,C 180.0000} C_DIS
LIN  {X -51.0000,Y 0.0000,Z 62.2754,A 180.0000,B 0.0000,C 180.0000} C_DIS
CIRC {X 0.0000,Y -51.0000,Z 62.2754,A 180.0000,B 0.0000,C 180.0000},{X 51.0000,Y 0.0000,Z 62.2754,A 180.0000,B 0.0000,C 180.0000} C_DIS
CIRC {X 0.0000,Y 51.0000,Z 62.2754,A 180.0000,B 0.0000,C 180.0000},{X -51.0000,Y 0.0000,Z 62.2754,A 180.0000,B 0.0000,C 180.0000} C_DIS
LIN  {X -51.0000,Y 0.0000,Z 62.8743,A 180.0000,B 0.0000,C 180.0000} C_DIS
CIRC {X 0.0000,Y -51.0000,Z 62.8743,A 180.0000,B 0.0000,C 180.0000},{X 51.0000,Y 0.0000,Z 62.8743,A 180.0000,B 0.0000,C 180.0000} C_DIS
CIRC {X 0.0000,Y 51.0000,Z 62.8743,A 180.0000,B 0.0000,C 180.0000},{X -51.0000,Y 0.0000,Z 62.8743,A 180.0000,B 0.0000,C 180.0000} C_DIS
LIN  {X -51.0000,Y 0.0000,Z 63.4731,A 180.0000,B 0.0000,C 180.0000} C_DIS
CIRC {X 0.0000,Y -51.0000,Z 63.4731,A 180.0000,B 0.0000,C 180.0000},{X 51.0000,Y 0.0000,Z 63.4731,A 180.0000,B 0.0000,C 180.0000} C_DIS
CIRC {X 0.0000,Y 51.0000,Z 63.4731,A 180.0000,B 0.0000,C 180.0000},{X -51.0000,Y 0.0000,Z 63.4731,A 180.0000,B 0.0000,C 180.0000} C_DIS
LIN  {X -51.0000,Y 0.0000,Z 64.0719,A 180.0000,B 0.0000,C 180.0000} C_DIS
CIRC {X 0.0000,Y -51.0000,Z 64.0719,A 180.0000,B 0.0000,C 180.0000},{X 51.0000,Y 0.0000,Z 64.0719,A 180.0000,B 0.0000,C 180.0000} C_DIS
CIRC {X 0.0000,Y 51.0000,Z 64.0719,A 180.0000,B 0.0000,C 180.0000},{X -51.0000,Y 0.0000,Z 64.0719,A 180.0000,B 0.0000,C 180.0000} C_DIS
LIN  {X -51.0000,Y 0.0000,Z 64.6707,A 180.0000,B 0.0000,C 180.0000} C_DIS
CIRC {X 0.0000,Y -51.0000,Z 64.6707,A 180.0000,B 0.0000,C 180.0000},{X 51.0000,Y 0.0000,Z 64.6707,A 180.0000,B 0.0000,C 180.0000} C_DIS
CIRC {X 0.0000,Y 51.0000,Z 64.6707,A 180.0000,B 0.0000,C 180.0000},{X -51.0000,Y 0.0000,Z 64.6707,A 180.0000,B 0.0000,C 180.0000} C_DIS
LIN  {X -51.0000,Y 0.0000,Z 65.2695,A 180.0000,B 0.0000,C 180.0000} C_DIS
CIRC {X 0.0000,Y -51.0000,Z 65.2695,A 180.0000,B 0.0000,C 180.0000},{X 51.0000,Y 0.0000,Z 65.2695,A 180.0000,B 0.0000,C 180.0000} C_DIS
CIRC {X 0.0000,Y 51.0000,Z 65.2695,A 180.0000,B 0.0000,C 180.0000},{X -51.0000,Y 0.0000,Z 65.2695,A 180.0000,B 0.0000,C 180.0000} C_DIS
LIN  {X -51.0000,Y 0.0000,Z 65.8683,A 180.0000,B 0.0000,C 180.0000} C_DIS
CIRC {X 0.0000,Y -51.0000,Z 65.8683,A 180.0000,B 0.0000,C 180.0000},{X 51.0000,Y 0.0000,Z 65.8683,A 180.0000,B 0.0000,C 180.0000} C_DIS
CIRC {X 0.0000,Y 51.0000,Z 65.8683,A 180.0000,B 0.0000,C 180.0000},{X -51.0000,Y 0.0000,Z 65.8683,A 180.0000,B 0.0000,C 180.0000} C_DIS
LIN  {X -51.0000,Y 0.0000,Z 66.4671,A 180.0000,B 0.0000,C 180.0000} C_DIS
CIRC {X 0.0000,Y -51.0000,Z 66.4671,A 180.0000,B 0.0000,C 180.0000},{X 51.0000,Y 0.0000,Z 66.4671,A 180.0000,B 0.0000,C 180.0000} C_DIS
CIRC {X 0.0000,Y 51.0000,Z 66.4671,A 180.0000,B 0.0000,C 180.0000},{X -51.0000,Y 0.0000,Z 66.4671,A 180.0000,B 0.0000,C 180.0000} C_DIS
LIN  {X -51.0000,Y 0.0000,Z 67.0659,A 180.0000,B 0.0000,C 180.0000} C_DIS
CIRC {X 0.0000,Y -51.0000,Z 67.0659,A 180.0000,B 0.0000,C 180.0000},{X 51.0000,Y 0.0000,Z 67.0659,A 180.0000,B 0.0000,C 180.0000} C_DIS
CIRC {X 0.0000,Y 51.0000,Z 67.0659,A 180.0000,B 0.0000,C 180.0000},{X -51.0000,Y 0.0000,Z 67.0659,A 180.0000,B 0.0000,C 180.0000} C_DIS
LIN  {X -51.0000,Y 0.0000,Z 67.6647,A 180.0000,B 0.0000,C 180.0000} C_DIS
CIRC {X 0.0000,Y -51.0000,Z 67.6647,A 180.0000,B 0.0000,C 180.0000},{X 51.0000,Y 0.0000,Z 67.6647,A 180.0000,B 0.0000,C 180.0000} C_DIS
CIRC {X 0.0000,Y 51.0000,Z 67.6647,A 180.0000,B 0.0000,C 180.0000},{X -51.0000,Y 0.0000,Z 67.6647,A 180.0000,B 0.0000,C 180.0000} C_DIS
LIN  {X -51.0000,Y 0.0000,Z 68.2635,A 180.0000,B 0.0000,C 180.0000} C_DIS
CIRC {X 0.0000,Y -51.0000,Z 68.2635,A 180.0000,B 0.0000,C 180.0000},{X 51.0000,Y 0.0000,Z 68.2635,A 180.0000,B 0.0000,C 180.0000} C_DIS
CIRC {X 0.0000,Y 51.0000,Z 68.2635,A 180.0000,B 0.0000,C 180.0000},{X -51.0000,Y 0.0000,Z 68.2635,A 180.0000,B 0.0000,C 180.0000} C_DIS
LIN  {X -51.0000,Y 0.0000,Z 68.8623,A 180.0000,B 0.0000,C 180.0000} C_DIS
CIRC {X 0.0000,Y -51.0000,Z 68.8623,A 180.0000,B 0.0000,C 180.0000},{X 51.0000,Y 0.0000,Z 68.8623,A 180.0000,B 0.0000,C 180.0000} C_DIS
CIRC {X 0.0000,Y 51.0000,Z 68.8623,A 180.0000,B 0.0000,C 180.0000},{X -51.0000,Y 0.0000,Z 68.8623,A 180.0000,B 0.0000,C 180.0000} C_DIS
LIN  {X -51.0000,Y 0.0000,Z 69.4611,A 180.0000,B 0.0000,C 180.0000} C_DIS
CIRC {X 0.0000,Y -51.0000,Z 69.4611,A 180.0000,B 0.0000,C 180.0000},{X 51.0000,Y 0.0000,Z 69.4611,A 180.0000,B 0.0000,C 180.0000} C_DIS
CIRC {X 0.0000,Y 51.0000,Z 69.4611,A 180.0000,B 0.0000,C 180.0000},{X -51.0000,Y 0.0000,Z 69.4611,A 180.0000,B 0.0000,C 180.0000} C_DIS
LIN  {X -51.0000,Y 0.0000,Z 70.0599,A 180.0000,B 0.0000,C 180.0000} C_DIS
CIRC {X 0.0000,Y -51.0000,Z 70.0599,A 180.0000,B 0.0000,C 180.0000},{X 51.0000,Y 0.0000,Z 70.0599,A 180.0000,B 0.0000,C 180.0000} C_DIS
CIRC {X 0.0000,Y 51.0000,Z 70.0599,A 180.0000,B 0.0000,C 180.0000},{X -51.0000,Y 0.0000,Z 70.0599,A 180.0000,B 0.0000,C 180.0000} C_DIS
LIN  {X -51.0000,Y 0.0000,Z 70.6587,A 180.0000,B 0.0000,C 180.0000} C_DIS
CIRC {X 0.0000,Y -51.0000,Z 70.6587,A 180.0000,B 0.0000,C 180.0000},{X 51.0000,Y 0.0000,Z 70.6587,A 180.0000,B 0.0000,C 180.0000} C_DIS
CIRC {X 0.0000,Y 51.0000,Z 70.6587,A 180.0000,B 0.0000,C 180.0000},{X -51.0000,Y 0.0000,Z 70.6587,A 180.0000,B 0.0000,C 180.0000} C_DIS
LIN  {X -51.0000,Y 0.0000,Z 71.2575,A 180.0000,B 0.0000,C 180.0000} C_DIS
CIRC {X 0.0000,Y -51.0000,Z 71.2575,A 180.0000,B 0.0000,C 180.0000},{X 51.0000,Y 0.0000,Z 71.2575,A 180.0000,B 0.0000,C 180.0000} C_DIS
CIRC {X 0.0000,Y 51.0000,Z 71.2575,A 180.0000,B 0.0000,C 180.0000},{X -51.0000,Y 0.0000,Z 71.2575,A 180.0000,B 0.0000,C 180.0000} C_DIS
LIN  {X -51.0000,Y 0.0000,Z 71.8563,A 180.0000,B 0.0000,C 180.0000} C_DIS
CIRC {X 0.0000,Y -51.0000,Z 71.8563,A 180.0000,B 0.0000,C 180.0000},{X 51.0000,Y 0.0000,Z 71.8563,A 180.0000,B 0.0000,C 180.0000} C_DIS
CIRC {X 0.0000,Y 51.0000,Z 71.8563,A 180.0000,B 0.0000,C 180.0000},{X -51.0000,Y 0.0000,Z 71.8563,A 180.0000,B 0.0000,C 180.0000} C_DIS
LIN  {X -51.0000,Y 0.0000,Z 72.4551,A 180.0000,B 0.0000,C 180.0000} C_DIS
CIRC {X 0.0000,Y -51.0000,Z 72.4551,A 180.0000,B 0.0000,C 180.0000},{X 51.0000,Y 0.0000,Z 72.4551,A 180.0000,B 0.0000,C 180.0000} C_DIS
CIRC {X 0.0000,Y 51.0000,Z 72.4551,A 180.0000,B 0.0000,C 180.0000},{X -51.0000,Y 0.0000,Z 72.4551,A 180.0000,B 0.0000,C 180.0000} C_DIS
LIN  {X -51.0000,Y 0.0000,Z 73.0539,A 180.0000,B 0.0000,C 180.0000} C_DIS
CIRC {X 0.0000,Y -51.0000,Z 73.0539,A 180.0000,B 0.0000,C 180.0000},{X 51.0000,Y 0.0000,Z 73.0539,A 180.0000,B 0.0000,C 180.0000} C_DIS
CIRC {X 0.0000,Y 51.0000,Z 73.0539,A 180.0000,B 0.0000,C 180.0000},{X -51.0000,Y 0.0000,Z 73.0539,A 180.0000,B 0.0000,C 180.0000} C_DIS
LIN  {X -51.0000,Y 0.0000,Z 73.6527,A 180.0000,B 0.0000,C 180.0000} C_DIS
CIRC {X 0.0000,Y -51.0000,Z 73.6527,A 180.0000,B 0.0000,C 180.0000},{X 51.0000,Y 0.0000,Z 73.6527,A 180.0000,B 0.0000,C 180.0000} C_DIS
CIRC {X 0.0000,Y 51.0000,Z 73.6527,A 180.0000,B 0.0000,C 180.0000},{X -51.0000,Y 0.0000,Z 73.6527,A 180.0000,B 0.0000,C 180.0000} C_DIS
LIN  {X -51.0000,Y 0.0000,Z 74.2515,A 180.0000,B 0.0000,C 180.0000} C_DIS
CIRC {X 0.0000,Y -51.0000,Z 74.2515,A 180.0000,B 0.0000,C 180.0000},{X 51.0000,Y 0.0000,Z 74.2515,A 180.0000,B 0.0000,C 180.0000} C_DIS
CIRC {X 0.0000,Y 51.0000,Z 74.2515,A 180.0000,B 0.0000,C 180.0000},{X -51.0000,Y 0.0000,Z 74.2515,A 180.0000,B 0.0000,C 180.0000} C_DIS
LIN  {X -51.0000,Y 0.0000,Z 74.8503,A 180.0000,B 0.0000,C 180.0000} C_DIS
CIRC {X 0.0000,Y -51.0000,Z 74.8503,A 180.0000,B 0.0000,C 180.0000},{X 51.0000,Y 0.0000,Z 74.8503,A 180.0000,B 0.0000,C 180.0000} C_DIS
CIRC {X 0.0000,Y 51.0000,Z 74.8503,A 180.0000,B 0.0000,C 180.0000},{X -51.0000,Y 0.0000,Z 74.8503,A 180.0000,B 0.0000,C 180.0000} C_DIS
LIN  {X -51.0000,Y 0.0000,Z 75.4491,A 180.0000,B 0.0000,C 180.0000} C_DIS
CIRC {X 0.0000,Y -51.0000,Z 75.4491,A 180.0000,B 0.0000,C 180.0000},{X 51.0000,Y 0.0000,Z 75.4491,A 180.0000,B 0.0000,C 180.0000} C_DIS
CIRC {X 0.0000,Y 51.0000,Z 75.4491,A 180.0000,B 0.0000,C 180.0000},{X -51.0000,Y 0.0000,Z 75.4491,A 180.0000,B 0.0000,C 180.0000} C_DIS
LIN  {X -51.0000,Y 0.0000,Z 76.0479,A 180.0000,B 0.0000,C 180.0000} C_DIS
CIRC {X 0.0000,Y -51.0000,Z 76.0479,A 180.0000,B 0.0000,C 180.0000},{X 51.0000,Y 0.0000,Z 76.0479,A 180.0000,B 0.0000,C 180.0000} C_DIS
CIRC {X 0.0000,Y 51.0000,Z 76.0479,A 180.0000,B 0.0000,C 180.0000},{X -51.0000,Y 0.0000,Z 76.0479,A 180.0000,B 0.0000,C 180.0000} C_DIS
LIN  {X -51.0000,Y 0.0000,Z 76.6467,A 180.0000,B 0.0000,C 180.0000} C_DIS
CIRC {X 0.0000,Y -51.0000,Z 76.6467,A 180.0000,B 0.0000,C 180.0000},{X 51.0000,Y 0.0000,Z 76.6467,A 180.0000,B 0.0000,C 180.0000} C_DIS
CIRC {X 0.0000,Y 51.0000,Z 76.6467,A 180.0000,B 0.0000,C 180.0000},{X -51.0000,Y 0.0000,Z 76.6467,A 180.0000,B 0.0000,C 180.0000} C_DIS
LIN  {X -51.0000,Y 0.0000,Z 77.2455,A 180.0000,B 0.0000,C 180.0000} C_DIS
CIRC {X 0.0000,Y -51.0000,Z 77.2455,A 180.0000,B 0.0000,C 180.0000},{X 51.0000,Y 0.0000,Z 77.2455,A 180.0000,B 0.0000,C 180.0000} C_DIS
CIRC {X 0.0000,Y 51.0000,Z 77.2455,A 180.0000,B 0.0000,C 180.0000},{X -51.0000,Y 0.0000,Z 77.2455,A 180.0000,B 0.0000,C 180.0000} C_DIS
LIN  {X -51.0000,Y 0.0000,Z 77.8443,A 180.0000,B 0.0000,C 180.0000} C_DIS
CIRC {X 0.0000,Y -51.0000,Z 77.8443,A 180.0000,B 0.0000,C 180.0000},{X 51.0000,Y 0.0000,Z 77.8443,A 180.0000,B 0.0000,C 180.0000} C_DIS
CIRC {X 0.0000,Y 51.0000,Z 77.8443,A 180.0000,B 0.0000,C 180.0000},{X -51.0000,Y 0.0000,Z 77.8443,A 180.0000,B 0.0000,C 180.0000} C_DIS
LIN  {X -51.0000,Y 0.0000,Z 78.4431,A 180.0000,B 0.0000,C 180.0000} C_DIS
CIRC {X 0.0000,Y -51.0000,Z 78.4431,A 180.0000,B 0.0000,C 180.0000},{X 51.0000,Y 0.0000,Z 78.4431,A 180.0000,B 0.0000,C 180.0000} C_DIS
CIRC {X 0.0000,Y 51.0000,Z 78.4431,A 180.0000,B 0.0000,C 180.0000},{X -51.0000,Y 0.0000,Z 78.4431,A 180.0000,B 0.0000,C 180.0000} C_DIS
LIN  {X -51.0000,Y 0.0000,Z 79.0419,A 180.0000,B 0.0000,C 180.0000} C_DIS
CIRC {X 0.0000,Y -51.0000,Z 79.0419,A 180.0000,B 0.0000,C 180.0000},{X 51.0000,Y 0.0000,Z 79.0419,A 180.0000,B 0.0000,C 180.0000} C_DIS
CIRC {X 0.0000,Y 51.0000,Z 79.0419,A 180.0000,B 0.0000,C 180.0000},{X -51.0000,Y 0.0000,Z 79.0419,A 180.0000,B 0.0000,C 180.0000} C_DIS
LIN  {X -51.0000,Y 0.0000,Z 79.6407,A 180.0000,B 0.0000,C 180.0000} C_DIS
CIRC {X 0.0000,Y -51.0000,Z 79.6407,A 180.0000,B 0.0000,C 180.0000},{X 51.0000,Y 0.0000,Z 79.6407,A 180.0000,B 0.0000,C 180.0000} C_DIS
CIRC {X 0.0000,Y 51.0000,Z 79.6407,A 180.0000,B 0.0000,C 180.0000},{X -51.0000,Y 0.0000,Z 79.6407,A 180.0000,B 0.0000,C 180.0000} C_DIS
LIN  {X -51.0000,Y 0.0000,Z 80.2395,A 180.0000,B 0.0000,C 180.0000} C_DIS
CIRC {X 0.0000,Y -51.0000,Z 80.2395,A 180.0000,B 0.0000,C 180.0000},{X 51.0000,Y 0.0000,Z 80.2395,A 180.0000,B 0.0000,C 180.0000} C_DIS
CIRC {X 0.0000,Y 51.0000,Z 80.2395,A 180.0000,B 0.0000,C 180.0000},{X -51.0000,Y 0.0000,Z 80.2395,A 180.0000,B 0.0000,C 180.0000} C_DIS
LIN  {X -51.0000,Y 0.0000,Z 80.8383,A 180.0000,B 0.0000,C 180.0000} C_DIS
CIRC {X 0.0000,Y -51.0000,Z 80.8383,A 180.0000,B 0.0000,C 180.0000},{X 51.0000,Y 0.0000,Z 80.8383,A 180.0000,B 0.0000,C 180.0000} C_DIS
CIRC {X 0.0000,Y 51.0000,Z 80.8383,A 180.0000,B 0.0000,C 180.0000},{X -51.0000,Y 0.0000,Z 80.8383,A 180.0000,B 0.0000,C 180.0000} C_DIS
LIN  {X -51.0000,Y 0.0000,Z 81.4371,A 180.0000,B 0.0000,C 180.0000} C_DIS
CIRC {X 0.0000,Y -51.0000,Z 81.4371,A 180.0000,B 0.0000,C 180.0000},{X 51.0000,Y 0.0000,Z 81.4371,A 180.0000,B 0.0000,C 180.0000} C_DIS
CIRC {X 0.0000,Y 51.0000,Z 81.4371,A 180.0000,B 0.0000,C 180.0000},{X -51.0000,Y 0.0000,Z 81.4371,A 180.0000,B 0.0000,C 180.0000} C_DIS
LIN  {X -51.0000,Y 0.0000,Z 82.0359,A 180.0000,B 0.0000,C 180.0000} C_DIS
CIRC {X 0.0000,Y -51.0000,Z 82.0359,A 180.0000,B 0.0000,C 180.0000},{X 51.0000,Y 0.0000,Z 82.0359,A 180.0000,B 0.0000,C 180.0000} C_DIS
CIRC {X 0.0000,Y 51.0000,Z 82.0359,A 180.0000,B 0.0000,C 180.0000},{X -51.0000,Y 0.0000,Z 82.0359,A 180.0000,B 0.0000,C 180.0000} C_DIS
LIN  {X -51.0000,Y 0.0000,Z 82.6347,A 180.0000,B 0.0000,C 180.0000} C_DIS
CIRC {X 0.0000,Y -51.0000,Z 82.6347,A 180.0000,B 0.0000,C 180.0000},{X 51.0000,Y 0.0000,Z 82.6347,A 180.0000,B 0.0000,C 180.0000} C_DIS
CIRC {X 0.0000,Y 51.0000,Z 82.6347,A 180.0000,B 0.0000,C 180.0000},{X -51.0000,Y 0.0000,Z 82.6347,A 180.0000,B 0.0000,C 180.0000} C_DIS
LIN  {X -51.0000,Y 0.0000,Z 83.2335,A 180.0000,B 0.0000,C 180.0000} C_DIS
CIRC {X 0.0000,Y -51.0000,Z 83.2335,A 180.0000,B 0.0000,C 180.0000},{X 51.0000,Y 0.0000,Z 83.2335,A 180.0000,B 0.0000,C 180.0000} C_DIS
CIRC {X 0.0000,Y 51.0000,Z 83.2335,A 180.0000,B 0.0000,C 180.0000},{X -51.0000,Y 0.0000,Z 83.2335,A 180.0000,B 0.0000,C 180.0000} C_DIS
LIN  {X -51.0000,Y 0.0000,Z 83.8323,A 180.0000,B 0.0000,C 180.0000} C_DIS
CIRC {X 0.0000,Y -51.0000,Z 83.8323,A 180.0000,B 0.0000,C 180.0000},{X 51.0000,Y 0.0000,Z 83.8323,A 180.0000,B 0.0000,C 180.0000} C_DIS
CIRC {X 0.0000,Y 51.0000,Z 83.8323,A 180.0000,B 0.0000,C 180.0000},{X -51.0000,Y 0.0000,Z 83.8323,A 180.0000,B 0.0000,C 180.0000} C_DIS
LIN  {X -51.0000,Y 0.0000,Z 84.4311,A 180.0000,B 0.0000,C 180.0000} C_DIS
CIRC {X 0.0000,Y -51.0000,Z 84.4311,A 180.0000,B 0.0000,C 180.0000},{X 51.0000,Y 0.0000,Z 84.4311,A 180.0000,B 0.0000,C 180.0000} C_DIS
CIRC {X 0.0000,Y 51.0000,Z 84.4311,A 180.0000,B 0.0000,C 180.0000},{X -51.0000,Y 0.0000,Z 84.4311,A 180.0000,B 0.0000,C 180.0000} C_DIS
LIN  {X -51.0000,Y 0.0000,Z 85.0299,A 180.0000,B 0.0000,C 180.0000} C_DIS
CIRC {X 0.0000,Y -51.0000,Z 85.0299,A 180.0000,B 0.0000,C 180.0000},{X 51.0000,Y 0.0000,Z 85.0299,A 180.0000,B 0.0000,C 180.0000} C_DIS
CIRC {X 0.0000,Y 51.0000,Z 85.0299,A 180.0000,B 0.0000,C 180.0000},{X -51.0000,Y 0.0000,Z 85.0299,A 180.0000,B 0.0000,C 180.0000} C_DIS
LIN  {X -51.0000,Y 0.0000,Z 85.6287,A 180.0000,B 0.0000,C 180.0000} C_DIS
CIRC {X 0.0000,Y -51.0000,Z 85.6287,A 180.0000,B 0.0000,C 180.0000},{X 51.0000,Y 0.0000,Z 85.6287,A 180.0000,B 0.0000,C 180.0000} C_DIS
CIRC {X 0.0000,Y 51.0000,Z 85.6287,A 180.0000,B 0.0000,C 180.0000},{X -51.0000,Y 0.0000,Z 85.6287,A 180.0000,B 0.0000,C 180.0000} C_DIS
LIN  {X -51.0000,Y 0.0000,Z 86.2275,A 180.0000,B 0.0000,C 180.0000} C_DIS
CIRC {X 0.0000,Y -51.0000,Z 86.2275,A 180.0000,B 0.0000,C 180.0000},{X 51.0000,Y 0.0000,Z 86.2275,A 180.0000,B 0.0000,C 180.0000} C_DIS
CIRC {X 0.0000,Y 51.0000,Z 86.2275,A 180.0000,B 0.0000,C 180.0000},{X -51.0000,Y 0.0000,Z 86.2275,A 180.0000,B 0.0000,C 180.0000} C_DIS
LIN  {X -51.0000,Y 0.0000,Z 86.8263,A 180.0000,B 0.0000,C 180.0000} C_DIS
CIRC {X 0.0000,Y -51.0000,Z 86.8263,A 180.0000,B 0.0000,C 180.0000},{X 51.0000,Y 0.0000,Z 86.8263,A 180.0000,B 0.0000,C 180.0000} C_DIS
CIRC {X 0.0000,Y 51.0000,Z 86.8263,A 180.0000,B 0.0000,C 180.0000},{X -51.0000,Y 0.0000,Z 86.8263,A 180.0000,B 0.0000,C 180.0000} C_DIS
LIN  {X -51.0000,Y 0.0000,Z 87.4252,A 180.0000,B 0.0000,C 180.0000} C_DIS
CIRC {X 0.0000,Y -51.0000,Z 87.4252,A 180.0000,B 0.0000,C 180.0000},{X 51.0000,Y 0.0000,Z 87.4252,A 180.0000,B 0.0000,C 180.0000} C_DIS
CIRC {X 0.0000,Y 51.0000,Z 87.4252,A 180.0000,B 0.0000,C 180.0000},{X -51.0000,Y 0.0000,Z 87.4252,A 180.0000,B 0.0000,C 180.0000} C_DIS
LIN  {X -51.0000,Y 0.0000,Z 88.0240,A 180.0000,B 0.0000,C 180.0000} C_DIS
CIRC {X 0.0000,Y -51.0000,Z 88.0240,A 180.0000,B 0.0000,C 180.0000},{X 51.0000,Y 0.0000,Z 88.0240,A 180.0000,B 0.0000,C 180.0000} C_DIS
CIRC {X 0.0000,Y 51.0000,Z 88.0240,A 180.0000,B 0.0000,C 180.0000},{X -51.0000,Y 0.0000,Z 88.0240,A 180.0000,B 0.0000,C 180.0000} C_DIS
LIN  {X -51.0000,Y 0.0000,Z 88.6228,A 180.0000,B 0.0000,C 180.0000} C_DIS
CIRC {X 0.0000,Y -51.0000,Z 88.6228,A 180.0000,B 0.0000,C 180.0000},{X 51.0000,Y 0.0000,Z 88.6228,A 180.0000,B 0.0000,C 180.0000} C_DIS
CIRC {X 0.0000,Y 51.0000,Z 88.6228,A 180.0000,B 0.0000,C 180.0000},{X -51.0000,Y 0.0000,Z 88.6228,A 180.0000,B 0.0000,C 180.0000} C_DIS
LIN  {X -51.0000,Y 0.0000,Z 89.2216,A 180.0000,B 0.0000,C 180.0000} C_DIS
CIRC {X 0.0000,Y -51.0000,Z 89.2216,A 180.0000,B 0.0000,C 180.0000},{X 51.0000,Y 0.0000,Z 89.2216,A 180.0000,B 0.0000,C 180.0000} C_DIS
CIRC {X 0.0000,Y 51.0000,Z 89.2216,A 180.0000,B 0.0000,C 180.0000},{X -51.0000,Y 0.0000,Z 89.2216,A 180.0000,B 0.0000,C 180.0000} C_DIS
LIN  {X -51.0000,Y 0.0000,Z 89.8204,A 180.0000,B 0.0000,C 180.0000} C_DIS
CIRC {X 0.0000,Y -51.0000,Z 89.8204,A 180.0000,B 0.0000,C 180.0000},{X 51.0000,Y 0.0000,Z 89.8204,A 180.0000,B 0.0000,C 180.0000} C_DIS
CIRC {X 0.0000,Y 51.0000,Z 89.8204,A 180.0000,B 0.0000,C 180.0000},{X -51.0000,Y 0.0000,Z 89.8204,A 180.0000,B 0.0000,C 180.0000} C_DIS
LIN  {X -51.0000,Y 0.0000,Z 90.4192,A 180.0000,B 0.0000,C 180.0000} C_DIS
CIRC {X 0.0000,Y -51.0000,Z 90.4192,A 180.0000,B 0.0000,C 180.0000},{X 51.0000,Y 0.0000,Z 90.4192,A 180.0000,B 0.0000,C 180.0000} C_DIS
CIRC {X 0.0000,Y 51.0000,Z 90.4192,A 180.0000,B 0.0000,C 180.0000},{X -51.0000,Y 0.0000,Z 90.4192,A 180.0000,B 0.0000,C 180.0000} C_DIS
LIN  {X -51.0000,Y 0.0000,Z 91.0180,A 180.0000,B 0.0000,C 180.0000} C_DIS
CIRC {X 0.0000,Y -51.0000,Z 91.0180,A 180.0000,B 0.0000,C 180.0000},{X 51.0000,Y 0.0000,Z 91.0180,A 180.0000,B 0.0000,C 180.0000} C_DIS
CIRC {X 0.0000,Y 51.0000,Z 91.0180,A 180.0000,B 0.0000,C 180.0000},{X -51.0000,Y 0.0000,Z 91.0180,A 180.0000,B 0.0000,C 180.0000} C_DIS
LIN  {X -51.0000,Y 0.0000,Z 91.6168,A 180.0000,B 0.0000,C 180.0000} C_DIS
CIRC {X 0.0000,Y -51.0000,Z 91.6168,A 180.0000,B 0.0000,C 180.0000},{X 51.0000,Y 0.0000,Z 91.6168,A 180.0000,B 0.0000,C 180.0000} C_DIS
CIRC {X 0.0000,Y 51.0000,Z 91.6168,A 180.0000,B 0.0000,C 180.0000},{X -51.0000,Y 0.0000,Z 91.6168,A 180.0000,B 0.0000,C 180.0000} C_DIS
LIN  {X -51.0000,Y 0.0000,Z 92.2156,A 180.0000,B 0.0000,C 180.0000} C_DIS
CIRC {X 0.0000,Y -51.0000,Z 92.2156,A 180.0000,B 0.0000,C 180.0000},{X 51.0000,Y 0.0000,Z 92.2156,A 180.0000,B 0.0000,C 180.0000} C_DIS
CIRC {X 0.0000,Y 51.0000,Z 92.2156,A 180.0000,B 0.0000,C 180.0000},{X -51.0000,Y 0.0000,Z 92.2156,A 180.0000,B 0.0000,C 180.0000} C_DIS
LIN  {X -51.0000,Y 0.0000,Z 92.8144,A 180.0000,B 0.0000,C 180.0000} C_DIS
CIRC {X 0.0000,Y -51.0000,Z 92.8144,A 180.0000,B 0.0000,C 180.0000},{X 51.0000,Y 0.0000,Z 92.8144,A 180.0000,B 0.0000,C 180.0000} C_DIS
CIRC {X 0.0000,Y 51.0000,Z 92.8144,A 180.0000,B 0.0000,C 180.0000},{X -51.0000,Y 0.0000,Z 92.8144,A 180.0000,B 0.0000,C 180.0000} C_DIS
LIN  {X -51.0000,Y 0.0000,Z 93.4132,A 180.0000,B 0.0000,C 180.0000} C_DIS
CIRC {X 0.0000,Y -51.0000,Z 93.4132,A 180.0000,B 0.0000,C 180.0000},{X 51.0000,Y 0.0000,Z 93.4132,A 180.0000,B 0.0000,C 180.0000} C_DIS
CIRC {X 0.0000,Y 51.0000,Z 93.4132,A 180.0000,B 0.0000,C 180.0000},{X -51.0000,Y 0.0000,Z 93.4132,A 180.0000,B 0.0000,C 180.0000} C_DIS
LIN  {X -51.0000,Y 0.0000,Z 94.0120,A 180.0000,B 0.0000,C 180.0000} C_DIS
CIRC {X 0.0000,Y -51.0000,Z 94.0120,A 180.0000,B 0.0000,C 180.0000},{X 51.0000,Y 0.0000,Z 94.0120,A 180.0000,B 0.0000,C 180.0000} C_DIS
CIRC {X 0.0000,Y 51.0000,Z 94.0120,A 180.0000,B 0.0000,C 180.0000},{X -51.0000,Y 0.0000,Z 94.0120,A 180.0000,B 0.0000,C 180.0000} C_DIS
LIN  {X -51.0000,Y 0.0000,Z 94.6108,A 180.0000,B 0.0000,C 180.0000} C_DIS
CIRC {X 0.0000,Y -51.0000,Z 94.6108,A 180.0000,B 0.0000,C 180.0000},{X 51.0000,Y 0.0000,Z 94.6108,A 180.0000,B 0.0000,C 180.0000} C_DIS
CIRC {X 0.0000,Y 51.0000,Z 94.6108,A 180.0000,B 0.0000,C 180.0000},{X -51.0000,Y 0.0000,Z 94.6108,A 180.0000,B 0.0000,C 180.0000} C_DIS
LIN  {X -51.0000,Y 0.0000,Z 95.2096,A 180.0000,B 0.0000,C 180.0000} C_DIS
CIRC {X 0.0000,Y -51.0000,Z 95.2096,A 180.0000,B 0.0000,C 180.0000},{X 51.0000,Y 0.0000,Z 95.2096,A 180.0000,B 0.0000,C 180.0000} C_DIS
CIRC {X 0.0000,Y 51.0000,Z 95.2096,A 180.0000,B 0.0000,C 180.0000},{X -51.0000,Y 0.0000,Z 95.2096,A 180.0000,B 0.0000,C 180.0000} C_DIS
LIN  {X -51.0000,Y 0.0000,Z 95.8084,A 180.0000,B 0.0000,C 180.0000} C_DIS
CIRC {X 0.0000,Y -51.0000,Z 95.8084,A 180.0000,B 0.0000,C 180.0000},{X 51.0000,Y 0.0000,Z 95.8084,A 180.0000,B 0.0000,C 180.0000} C_DIS
CIRC {X 0.0000,Y 51.0000,Z 95.8084,A 180.0000,B 0.0000,C 180.0000},{X -51.0000,Y 0.0000,Z 95.8084,A 180.0000,B 0.0000,C 180.0000} C_DIS
LIN  {X -51.0000,Y 0.0000,Z 96.4072,A 180.0000,B 0.0000,C 180.0000} C_DIS
CIRC {X 0.0000,Y -51.0000,Z 96.4072,A 180.0000,B 0.0000,C 180.0000},{X 51.0000,Y 0.0000,Z 96.4072,A 180.0000,B 0.0000,C 180.0000} C_DIS
CIRC {X 0.0000,Y 51.0000,Z 96.4072,A 180.0000,B 0.0000,C 180.0000},{X -51.0000,Y 0.0000,Z 96.4072,A 180.0000,B 0.0000,C 180.0000} C_DIS
LIN  {X -51.0000,Y 0.0000,Z 97.0060,A 180.0000,B 0.0000,C 180.0000} C_DIS
CIRC {X 0.0000,Y -51.0000,Z 97.0060,A 180.0000,B 0.0000,C 180.0000},{X 51.0000,Y 0.0000,Z 97.0060,A 180.0000,B 0.0000,C 180.0000} C_DIS
CIRC {X 0.0000,Y 51.0000,Z 97.0060,A 180.0000,B 0.0000,C 180.0000},{X -51.0000,Y 0.0000,Z 97.0060,A 180.0000,B 0.0000,C 180.0000} C_DIS
LIN  {X -51.0000,Y 0.0000,Z 97.6048,A 180.0000,B 0.0000,C 180.0000} C_DIS
CIRC {X 0.0000,Y -51.0000,Z 97.6048,A 180.0000,B 0.0000,C 180.0000},{X 51.0000,Y 0.0000,Z 97.6048,A 180.0000,B 0.0000,C 180.0000} C_DIS
CIRC {X 0.0000,Y 51.0000,Z 97.6048,A 180.0000,B 0.0000,C 180.0000},{X -51.0000,Y 0.0000,Z 97.6048,A 180.0000,B 0.0000,C 180.0000} C_DIS
LIN  {X -51.0000,Y 0.0000,Z 98.2036,A 180.0000,B 0.0000,C 180.0000} C_DIS
CIRC {X 0.0000,Y -51.0000,Z 98.2036,A 180.0000,B 0.0000,C 180.0000},{X 51.0000,Y 0.0000,Z 98.2036,A 180.0000,B 0.0000,C 180.0000} C_DIS
CIRC {X 0.0000,Y 51.0000,Z 98.2036,A 180.0000,B 0.0000,C 180.0000},{X -51.0000,Y 0.0000,Z 98.2036,A 180.0000,B 0.0000,C 180.0000} C_DIS
LIN  {X -51.0000,Y 0.0000,Z 98.8024,A 180.0000,B 0.0000,C 180.0000} C_DIS
CIRC {X 0.0000,Y -51.0000,Z 98.8024,A 180.0000,B 0.0000,C 180.0000},{X 51.0000,Y 0.0000,Z 98.8024,A 180.0000,B 0.0000,C 180.0000} C_DIS
CIRC {X 0.0000,Y 51.0000,Z 98.8024,A 180.0000,B 0.0000,C 180.0000},{X -51.0000,Y 0.0000,Z 98.8024,A 180.0000,B 0.0000,C 180.0000} C_DIS
LIN  {X -51.0000,Y 0.0000,Z 99.4012,A 180.0000,B 0.0000,C 180.0000} C_DIS
CIRC {X 0.0000,Y -51.0000,Z 99.4012,A 180.0000,B 0.0000,C 180.0000},{X 51.0000,Y 0.0000,Z 99.4012,A 180.0000,B 0.0000,C 180.0000} C_DIS
CIRC {X 0.0000,Y 51.0000,Z 99.4012,A 180.0000,B 0.0000,C 180.0000},{X -51.0000,Y 0.0000,Z 99.4012,A 180.0000,B 0.0000,C 180.0000} C_DIS
LIN  {X -51.0000,Y 0.0000,Z 100.0000,A 180.0000,B 0.0000,C 180.0000} C_DIS
CIRC {X 0.0000,Y -51.0000,Z 100.0000,A 180.0000,B 0.0000,C 180.0000},{X 51.0000,Y 0.0000,Z 100.0000,A 180.0000,B 0.0000,C 180.0000} C_DIS
CIRC {X 0.0000,Y 51.0000,Z 100.0000,A 180.0000,B 0.0000,C 180.0000},{X -51.0000,Y 0.0000,Z 100.0000,A 180.0000,B 0.0000,C 180.0000} C_DIS
CIRC {X -56.8579,Y -14.1421,Z 100.0000,A 180.0000,B 0.0000,C 180.0000},{X -71.0000,Y -20.0000,Z 100.0000,A 180.0000,B 0.0000,C 180.0000} C_DIS
LIN  {X -91.0000,Y -20.0000,Z 100.0000,A 180.0000,B 0.0000,C 180.0000} C_DIS
PTP  {X -91.0000,Y -20.0000,Z 125.0000,A 180.0000,B 0.0000,C 180.0000,S 2,T 10}
PTP  {A1 20.0000,A2 -90.0000,A3 90.0000,A4 0.0000,A5 45.0000,A6 0.0000}

END
